(* CODESYS project OC_Profinet.library
   DefaultNamespace: OC_Profinet
   Description: Open Commissioning Library for Profinet devices
   Author: SpiraTec AG
   Title: OC_Profinet
   Version: 1.0.1
   Company: Open Commissioning
   Placeholder: OC_Profinet

Project tree, tasks and I/O mapping:
  libraries: OC_Core, * (Open Commissioning); OC_Profisafe, * (Open Commissioning); Tc2_Math, * (Beckhoff Automation GmbH); Tc2_Standard, * (Beckhoff Automation GmbH); Tc2_System, * (Beckhoff Automation GmbH); Tc2_Utilities, * (Beckhoff Automation GmbH); Tc3_Module, * (Beckhoff Automation GmbH); TcUnit, * (www.tcunit.org)
  Common/
    ProfidriveGSM/
      data type E_ProfidriveGSM_State
      function block FB_ProfidriveGSM [ST]: eState, S0_Disabled, S1_SwitchingOnInhibited, S2_ReadyForSwitchingOn, S3_SwitchedOn, S4_Operation, S51_RampStop, S52_QuickStop
      data type ST_ProfidriveGSM_Control
      data type ST_ProfidriveGSM_Status
    ProfidriveParamInterpreter/
      data type E_ProfidriveParam_Format
      function block FB_ProfidriveParamInterpreter [ST]: FormatSize, FormatType, MakeResponse, Reset
      data type ST_ProfidriveParam
      data type ST_ProfidriveParam_Set
    Utils/
      function F_CalcCrc16 [ST]
  Devices/
    Profidrive_Telegram1/
      function block FB_Profidrive_Telegram1 [ST]: Cycle, GetControlData, InitRun, Operation, SetStatusData
      data type ST_Profidrive_Telegram1_Config
      data type ST_Profidrive_Telegram1_Control
      data type ST_Profidrive_Telegram1_Status
    SEW_MoviC_Position/
      data type E_SEW_MoviC_Position_OperationMode
      function block FB_SEW_MoviC_Position [ST]: Cycle, GetControlData, InitRun, Operation, Safety, SetStatusData
      data type ST_SEW_MoviC_Position_Config
      data type ST_SEW_MoviC_Position_Control
      data type ST_SEW_MoviC_Position_Status
    SEW_MoviC_Velocity/
      function block FB_SEW_MoviC_Velocity [ST]: Cycle, GetControlData, InitRun, Operation, Safety, SetStatusData
      data type ST_SEW_MoviC_Velocity_Config
      data type ST_SEW_MoviC_Velocity_Control
      data type ST_SEW_MoviC_Velocity_Status
    SEW_Movisafe_CSSx1a/
      function block FB_SEW_Movisafe_CSSx1a [ST]: bSTO, Cycle, GetControlData, InitRun, SetStatusData
      data type ST_SEW_Movisafe_CSSx1a_Config
      data type ST_SEW_Movisafe_CSSx1a_Control
      data type ST_SEW_Movisafe_CSSx1a_Status
    Siemens_RcvDp/
      function block FB_Siemens_RcvDp [ST]: Cycle, GetControlData, InitRun, SetStatusData, SimLogic
      data type ST_Siemens_RcvDp_Config
      data type ST_Siemens_RcvDp_Control
      data type ST_Siemens_RcvDp_DevData
      data type ST_Siemens_RcvDp_HstData
      data type ST_Siemens_RcvDp_Status
    Siemens_SendDp/
      function block FB_Siemens_SendDp [ST]: Cycle, GetControlData, InitRun, SetStatusData, SimLogic
      data type ST_Siemens_SendDp_Config
      data type ST_Siemens_SendDp_Control
      data type ST_Siemens_SendDp_DevData
      data type ST_Siemens_SendDp_HstData
      data type ST_Siemens_SendDp_Status
    interface I_SEW_Movisafe: bSTO
*)

// Common/ProfidriveGSM/E_ProfidriveGSM_State
{attribute 'qualified_only'}
{attribute 'strict'}
{attribute 'conditionalshow'}
TYPE E_ProfidriveGSM_State :
(
	S0_Disabled := 0,
	S1_SwitchingOnInhibited := 1,
	S2_ReadyForSwitchingOn := 2,
	S3_SwitchedOn := 3,
	S4_Operation := 4,
	S51_RampStop := 51,
	S52_QuickStop := 52
);
END_TYPE

// Common/ProfidriveGSM/ST_ProfidriveGSM_Control
(*
	Steuerwort 1 (STW1)
	Steuerwort 1 SIEMENS Telegramm 10x
	https://cache.industry.siemens.com/dl/files/665/109770665/att_1023132/v2/109770665_PROFIdrive_Statemachine_DOC_V10_de.pdf
*)
{attribute 'pack_mode' := '1'}
TYPE ST_ProfidriveGSM_Control :
STRUCT
	b0_On 							: BIT; 	//ON/OFF (OFF1)
	b1_CoastStop					: BIT; 	//The axis will not coast stop if this bit is set (OFF2)
	b2_QuickStop					: BIT; 	//The axis will not execute quick stop if this bit is set. Quick stop executes a controlled stop on the axis. (OFF3)
	b3_EnableOperation				: BIT; 	//The axis will enable and execute command if all preconditions are set. If a Wake and Shake procedure has to be executed as part of enabling, the transition to state "S4: Operation Enabled" is delayed until the procedure is finished.
	b4_Reserve						: BIT;	//Reserve
	b5_Reserve						: BIT;	//Reserve
	b6_Reserve						: BIT;	//Reserve
	b7_FaultAcknowledge				: BIT;	//Set this bit to reset faults on the drive.
	b8_Reserve						: BIT;	//Reserve
	b9_Reserve						: BIT;	//Reserve	
	b10_ControlPlc					: BIT;	//When not set, no command is accepted from the PLC.	
	b11_Reserved					: BIT;	//Reserve
	b12_Reserved					: BIT;	//Reserve
	b13_Reserved					: BIT;	//Reserve
	b14_Reserved					: BIT;	//Reserve
	b15_Reserved					: BIT;	//Reserve
END_STRUCT
END_TYPE

// Common/ProfidriveGSM/ST_ProfidriveGSM_Status
(*
	Zustandswort 1 (ZSW1)
	Zustandswort 1 SIEMENS Telegramm 10x
	https://cache.industry.siemens.com/dl/files/665/109770665/att_1023132/v2/109770665_PROFIdrive_Statemachine_DOC_V10_de.pdf
*)

{attribute 'pack_mode' := '1'}
TYPE ST_ProfidriveGSM_Status :
STRUCT
	b0_ReadyToSwitchOn 				: BIT; 	//Ready to switch on
	b1_ReadyForOperation			: BIT; 	//Ready for operation
	b2_OperationEnabled				: BIT; 	//Operation enabled
	b3_FaultPresent					: BIT; 	//A fault is present on the axis
	b4_CoastStop 					: BIT;	//No coast stop is executed (No OFF2 is active)
	b5_QuickStop					: BIT;	//No quick stop is executed (No OFF3 is active)
	b6_SwitchingOnInhibited			: BIT;	//Switch-on inhibit Switching on again is only possible through OFF1 and subsequent ON.
	b7_WarningPresent				: BIT;	//Warning present. The drive is operating. No acknowledgment required
	b8_Reserve						: BIT;	//Reserve
	b9_ControlRequested				: BIT;	//Control requested by the master
	b10_Reserved					: BIT;	//Reserve
	b11_Reserved					: BIT;	//Reserve
	b12_Reserved					: BIT;	//Reserve
	b13_Reserved					: BIT;	//Reserve
	b14_Reserved					: BIT;	//Reserve
	b15_Reserved					: BIT;	//Reserve
END_STRUCT
END_TYPE

// Common/ProfidriveParamInterpreter/E_ProfidriveParam_Format
{attribute 'qualified_only'}
{attribute 'strict'}
{attribute 'conditionalshow'}
TYPE E_ProfidriveParam_Format :
(
	UNKNOWN := 0,
	INT8	:= 2,
	INT16	:= 3,
	INT32	:= 4,
	UINT8	:= 5,
	UINT16	:= 6,
	UINT32	:= 7,
	FLOAT	:= 8,
	ZERO	:= 64,
	BYTE_	:= 65,
	WORD_	:= 66,
	DWORD_	:= 67,
	ERROR	:= 68
) BYTE;
END_TYPE

// Common/ProfidriveParamInterpreter/ST_ProfidriveParam
{attribute 'conditionalshow'}
TYPE ST_ProfidriveParam :
STRUCT
	nAttribute	: BYTE;
	nNumber		: UINT;
	nSubIndex	: UINT;
	nElements	: BYTE;
	nFormat		: E_ProfidriveParam_Format;
	aValue		: ARRAY[0..234] OF BYTE;
END_STRUCT
END_TYPE

// Common/ProfidriveParamInterpreter/ST_ProfidriveParam_Set
{attribute 'conditionalshow'}
TYPE ST_ProfidriveParam_Set :
	ARRAY[0..22] OF ST_ProfidriveParam; 
END_TYPE

// Devices/Profidrive_Telegram1/ST_Profidrive_Telegram1_Config
TYPE ST_Profidrive_Telegram1_Config :
STRUCT
	bForceMode					: BOOL; //Ignore process data from fieldbus.
	bSwapProcessData			: BOOL; //Reverse process data byte order from/to fieldbus.
	fRampDownTimeCoastStop 		: REAL := 1.0;		//Coast stop deceleration time in s
	bControlRequested			: BOOL := TRUE;
	bOutputVelocity				: BOOL := TRUE;		//TRUE: TargetValue = Velocity, FALSE: TargetValue = Position
	fP1058						: REAL := 150.0;	//JOG 1 velocity in rotation/s
	fP1059						: REAL := -150.0;	//JOG 1 velocity in rotation/s
	fP1120						: REAL := 2.0;		//Default acceleration time in s
	fP1121						: REAL := 2.0;		//Default deceleration time in s
	fP1135						: REAL := 1.0;		//Ramp down time quick stop in s
	fP2000						: REAL := 3000;		//Velocity in rotation/s when targeting 16#4000
	nR0035						: REAL := 60.0; 	//Temperature in degree celcius	
END_STRUCT
END_TYPE

// Devices/Profidrive_Telegram1/ST_Profidrive_Telegram1_Control
TYPE ST_Profidrive_Telegram1_Control :
STRUCT
	b0_Off1								: BOOL;	//STW1_0	0 = OFF1 (braking with ramp-function generator, then pulse suppression & ready for switching on) | 0 → 1 = ON (pulses can be enabled)
	b1_Off2								: BOOL;	//STW1_1	0 = OFF2 (immediate pulse suppression and switching on inhibited) | 1 = No OFF2 (enable is possible)
	b2_Off3								: BOOL;	//STW1_2	0 = OFF3 (braking with the OFF3 ramp p1135, then pulse suppression and switching on inhibited) | 1 = No OFF3 (enable possible) 
	b3_EnableOperation					: BOOL;	//STW1_3	0 = Inhibit operation (suppress pulses) | 1 = Enable operation (pulses can be enabled) 
	b4_OperatingCondition				: BOOL;	//STW1_4	0 = Inhibit ramp-function generator (set the ramp-function generator output to zero) | 1 = Operating condition (the ramp-function generator can be enabled)
	b5_ContinueRampFunctionGenerator	: BOOL;	//STW1_5	0 = Freeze ramp-function generator (freeze the ramp-function generator output) | 1 = Continue ramp-function generator 
	b6_EnableSetpoint  					: BOOL;	//STW1_6	0 = Inhibit setpoint (set the ramp-function generator input to zero) | 1 = Enable setpoint 
	b7_AcknowledgeFaults				: BOOL;	//STW1_7	0 → 1: = Acknowledge faults	                            
	b8_Jog1								: BOOL;	//STW1_8	1 = Jog 1 signal source
	b9_Jog2								: BOOL;	//STW1_9	1 = Jog 2 signal source
	b10_ControlByPlc					: BOOL;	//STW1_10	1 = Control by PLC
	b11_SetpointInversion				: BOOL;	//STW1_11	1 = Setpoint inversion
	b12_Reserved						: BOOL;	//STW1_12	Reserved
	b13_PotentiometerSetpointRaise		: BOOL;	//STW1_13	1 = Motorized potentiometer setpoint raise
	b14_PotentiometerSetpointLower		: BOOL;	//STW1_14	1 = Motorized potentiometer setpoint lower
	b15_Reserved						: BOOL;	//STW1_15	Reserved	
	nTargetVelocity						: INT;
END_STRUCT
END_TYPE

// Devices/Profidrive_Telegram1/ST_Profidrive_Telegram1_Status
TYPE ST_Profidrive_Telegram1_Status :
STRUCT
	b0_ReadyForSwitchingOn				: BOOL; // ZSW1_0	1 = Ready for switching on
	b1_ReadyForOperation				: BOOL; // ZSW1_1	1 = Ready for operation
	b2_OperationEnabled					: BOOL; // ZSW1_2	1 = Operation enabled
	b3_FaultPresent						: BOOL; // ZSW1_3	1 = Fault present
	b4_NoCoastDownActive				: BOOL; // ZSW1_4	1 = No coast down active (OFF2 inactive)
	b5_NoQuickStopActive				: BOOL; // ZSW1_5	1 = No quick stop active (OFF3 inactive)
	b6_SwitchingOnInhibited				: BOOL; // ZSW1_6	1 = Switching on inhibited active
	b7_AlarmPresent						: BOOL; // ZSW1_7	1 = Alarm present                        	
	b8_DeviationWithinTolerance			: BOOL; // ZSW1_8	1 = Speed setpoint - actual value deviation within tolerance t_off
	b9_ControlRequested					: BOOL; // ZSW1_9	1 = Control requested        
	b10_RpmCompValueReachedOrExceeded	: BOOL; // ZSW1_10	1 = f or n comparison value reached/exceeded  
	b11_TorqueOrPowerLimitNotReached	: BOOL; // ZSW1_11	1 = I, M, or P limit not reached     
	b12_OpenHoldingBrake 				: BOOL; // ZSW1_12	1 = Open the holding brake      
	b13_NoOvertempAlarm					: BOOL; // ZSW1_13	1 = No motor overtemperature alarm      
	b14_MotorRotatesForwards			: BOOL; // ZSW1_14	1 = Motor rotates forwards (n_act >= 0) | 0 = Motor rotates backwards (n_act < 0)   
	b15_NoAlarmNoOvertempPowerUnit		: BOOL; // ZSW1_15	1 = No alarm, thermal overload, power unit  
	nVelocity							: INT;
END_STRUCT
END_TYPE

// Devices/SEW_MoviC_Position/E_SEW_MoviC_Position_OperationMode
{attribute 'qualified_only'}
TYPE E_SEW_MoviC_Position_OperationMode :
(
	Jog					:= 100, //Position controlled jogging
	JogNoEnc			:= 101, //Speed controlled jogging
	SpeedControl		:= 200, //Speed control
	ReferenceParam		:= 300, //Reference travel, offset via parameter
	ReferenceBus		:= 301, //Reference travel, offset via fieldbus
	PositionAbs			:= 400, //Absolute position control
	PositionRel			:= 401, //Relative position control
	PositionModPos		:= 402, //Modulo position control, positive
	PositionModNeg		:= 403, //Modulo position control, negative
	PositionModShort	:= 404, //Modulo position control, shortest distance
	EnergyOptimized		:= 1200, //Energieoptimiertes Positionieren
	MechanicsOptimized	:= 1210	 //Mechanikoptimiertes Positionieren
)INT;
END_TYPE

// Devices/SEW_MoviC_Position/ST_SEW_MoviC_Position_Config
TYPE ST_SEW_MoviC_Position_Config :
STRUCT
	bForceMode				: BOOL; //Ignore process data from fieldbus.
	bSwapProcessData		: BOOL; //Reverse process data byte order from/to fieldbus.
	nSoftwareLimitMin		: DINT := -2147483648;	//Position limit minimum in LU
	nSoftwareLimitMax		: DINT := 2147483647;	//Position limit maximum in LU
	nReferencePos			: DINT := 0;			//Reference position in LU when using mode 300
	fDecCoastStop			: REAL := 1000.0;		//Deceleration for coast/brake stop in LU/s^2
	fDecEstop				: REAL := 100.0;		//Deceleration for emergency stop in LU/s^2
	fDecelerationLimit		: REAL := 100.0;		//Decceleration limit (bus stop) in LU/s^2
	fRatioVelocity			: REAL := 1.0;			//Ratio for setpoint velocity
	fRatioAccDec			: REAL := 1.0;			//Ratio for setpoint acceleration/deceleration
	fRatioPosition			: REAL := 1.0;			//Ratio for position output
	nJerk					: INT  := 0;			//Jerk from 0 to 100%
	fPositionOffset			: REAL := 0;
	fInitPosition			: REAL := 0;
	fResolution				: REAL := 0.1;
END_STRUCT
END_TYPE

// Devices/SEW_MoviC_Position/ST_SEW_MoviC_Position_Control
{attribute 'pack_mode' := '1'}
TYPE ST_SEW_MoviC_Position_Control :
STRUCT
    b0_EnableEStop 					: BIT;	//0  1 = enable, 0 = emergency stop
    b1_EnableBusStop 				: BIT;	//1  1 = enable, 0 = stop at application limits
    b2_Reserved2 					: BIT;	//2
    b3_ReleaseBrake 				: BIT;	//3  only needed if function is activated
    b4_JoggingCW 					: BIT;	//4  jog positive
    b5_JoggingCCW 					: BIT;	//5  jog negative
    b6_AcceptRelativePosition 		: BIT;	//6  apply relative target pos only in relative pos mode
    b7_StartStop 					: BIT;	//7  1 = start movement in all modes except jog, 0 = deceleration to speed 0
    b8_ErrorReset 					: BIT;	//8  reset fault messages
    b9_Reserved9 					: BIT;	//9
    b10_ActivateDriveTrain2 		: BIT;	//10  0 = drive train 1 selected, 1 = drive train 2 selected
    b11_Reserved11 					: BIT;	//11
    b12_DisableSoftwareLimits 		: BIT;	//12  0 = software limit activated, 1 = software limit deactivated
    b13_ActivateInhibit 			: BIT;	//13  1 = output stage inhibit activated -> motor coasts to halt or brake is applied, 0 = output stage can be enabled
    b14_ActivateStandByMode 		: BIT;	//14  1 = activated, can only be activated when output stage is inhibited (bActivateInhibit = 1)
    b15_MovikitHeartbeat 			: BIT;	//15  Heartbeat trigger
	nSetpointSpeed					: INT;	//16..31 
	nSetpointAcceleration			: INT;	//32..47
	nSetpointDeceleration			: INT;	//48..63
	nDigitalOutputs					: WORD;	//64..79
	nTargetApplicationMode			: E_SEW_MoviC_Position_OperationMode; //80..95
	nTargetPosition					: DINT;	//96..127
END_STRUCT
END_TYPE

// Devices/SEW_MoviC_Position/ST_SEW_MoviC_Position_Status
{attribute 'pack_mode' := '1'}
TYPE ST_SEW_MoviC_Position_Status :
STRUCT
	b0_InverterReady					: BIT;	//0  1 = Ready
	b1_STOInactive						: BIT;	//1  1 = STO inactive
	b2_PowerStageOn						: BIT;	//2  1 = Output stage enable
	b3_BrakeReleased					: BIT;	//3  1 = Brake released
	b4_MotorTurning						: BIT;	//4  1 = Motor running
	b5_DriveReferenced					: BIT;	//5  1 = Active drive referenced
	b6_SetpointsActive					: BIT;	//6  1 = New relative position applied
	b7_TargetpositionReached			: BIT;	//7  1 = In position
	b8_ErrorActive						: BIT;	//8  1 = Fault
	b9_WarningActive					: BIT;	//9  1 = Warning
	b10_DriveTrain2Active				: BIT;	//10  1 = Drive train 2 active
	b11_SpeedSetpointReached			: BIT;	//11  1 = "Setpoint/actual speed comparison active" signal
	b12_SoftwareLimitsDisabled			: BIT;	//12  1 = Software limit switches inactive
	b13_OutputStageInhibit 				: BIT;	//13  1 = Output stage inhibit 
	b14_StandByModeActive				: BIT;	//14  1 = Standby mode active
	b15_MovikitHeartbeat				: BIT;	//15  Heartbeat trigger mirror
	nActualSpeed						: INT;	//16..31
	nActualStatus						: WORD;	//32..47
	nActualTorque						: INT;	//48..63
	nDigitalInputs						: WORD;	//64..79
	nActualApplicationMode				: E_SEW_MoviC_Position_OperationMode; //80..95
	nActualPosition						: DINT;	//96..127 
END_STRUCT
END_TYPE

// Devices/SEW_MoviC_Velocity/ST_SEW_MoviC_Velocity_Config
TYPE ST_SEW_MoviC_Velocity_Config :
STRUCT
	bForceMode				: BOOL; //Ignore process data from fieldbus.
	bSwapProcessData		: BOOL; //Reverse process data byte order from/to fieldbus.
	nSoftwareLimitMin		: DINT := -2147483648;	//Position limit minimum in LU
	nSoftwareLimitMax		: DINT := 2147483647;	//Position limit maximum in LU
	nReferencePos			: DINT := 0;			//Reference position in LU when using mode 300
	fDecCoastStop			: REAL := 1000.0;		//Deceleration for coast/brake stop in LU/s^2
	fDecEstop				: REAL := 100.0;		//Deceleration for emergency stop in LU/s^2
	fDecelerationLimit		: REAL := 100.0;		//Decceleration limit (bus stop) in LU/s^2
	fRatioVelocity			: REAL := 1.0;			//Ratio for setpoint velocity
	fRatioAccDec			: REAL := 1.0;			//Ratio for setpoint acceleration/deceleration
	fRatioPosition			: REAL := 1.0;			//Ratio for position output
	nJerk					: INT  := 0;			//Jerk from 0 to 100%
	fPositionOffset			: REAL := 0;
	fInitPosition			: REAL := 0;
	fResolution				: REAL := 0.1;
	bOutputVelocity			: BOOL := TRUE;			//TRUE: TargetValue = Velocity, FALSE: TargetValue = Position
END_STRUCT
END_TYPE

// Devices/SEW_MoviC_Velocity/ST_SEW_MoviC_Velocity_Control
TYPE ST_SEW_MoviC_Velocity_Control :
STRUCT
    b0_EnableEStop 					: BIT;	//0  1 = enable, 0 = emergency stop
    b1_EnableBusStop 				: BIT;	//1  1 = enable, 0 = stop at application limits
    b2_Reserved2 					: BIT;	//2
    b3_ReleaseBrake 				: BIT;	//3  only needed if function is activated
    b4_JoggingCW 					: BIT;	//4  jog positive
    b5_JoggingCCW 					: BIT;	//5  jog negative
    b6_AcceptRelativePosition 		: BIT;	//6  apply relative target pos only in relative pos mode
    b7_StartStop 					: BIT;	//7  1 = start movement in all modes except jog, 0 = deceleration to speed 0
    b8_ErrorReset 					: BIT;	//8  reset fault messages
    b9_Reserved9 					: BIT;	//9
    b10_ActivateDriveTrain2 		: BIT;	//10  0 = drive train 1 selected, 1 = drive train 2 selected
    b11_Reserved11 					: BIT;	//11
    b12_DisableSoftwareLimits 		: BIT;	//12  0 = software limit activated, 1 = software limit deactivated
    b13_ActivateInhibit 			: BIT;	//13  1 = output stage inhibit activated -> motor coasts to halt or brake is applied, 0 = output stage can be enabled
    b14_ActivateStandByMode 		: BIT;	//14  1 = activated, can only be activated when output stage is inhibited (bActivateInhibit = 1)
    b15_MovikitHeartbeat 			: BIT;	//15  Heartbeat trigger
	nSetpointSpeed					: INT;	//16..31 
	nSetpointAcceleration			: INT;	//32..47
	nSetpointDeceleration			: INT;	//48..63
	nDigitalOutputs					: WORD;	//64..79	
END_STRUCT
END_TYPE

// Devices/SEW_MoviC_Velocity/ST_SEW_MoviC_Velocity_Status
{attribute 'pack_mode' := '1'}
TYPE ST_SEW_MoviC_Velocity_Status :
STRUCT
	b0_InverterReady					: BIT;	//0  1 = Ready
	b1_STOInactive						: BIT;	//1  1 = STO inactive
	b2_PowerStageOn						: BIT;	//2  1 = Output stage enable
	b3_BrakeReleased					: BIT;	//3  1 = Brake released
	b4_MotorTurning						: BIT;	//4  1 = Motor running
	b5_DriveReferenced					: BIT;	//5  1 = Active drive referenced
	b6_SetpointsActive					: BIT;	//6  1 = New relative position applied
	b7_TargetpositionReached			: BIT;	//7  1 = In position
	b8_ErrorActive						: BIT;	//8  1 = Fault
	b9_WarningActive					: BIT;	//9  1 = Warning
	b10_DriveTrain2Active				: BIT;	//10  1 = Drive train 2 active
	b11_SpeedSetpointReached			: BIT;	//11  1 = "Setpoint/actual speed comparison active" signal
	b12_SoftwareLimitsDisabled			: BIT;	//12  1 = Software limit switches inactive
	b13_OutputStageInhibit 				: BIT;	//13  1 = Output stage inhibit 
	b14_StandByModeActive				: BIT;	//14  1 = Standby mode active
	b15_MovikitHeartbeat				: BIT;	//15  Heartbeat trigger mirror
	nActualSpeed						: INT;	//16..31
	nActualStatus						: WORD;	//32..47
	nActualTorque						: INT;	//48..63
	nDigitalInputs						: WORD;	//64..79	
END_STRUCT
END_TYPE

// Devices/SEW_Movisafe_CSSx1a/ST_SEW_Movisafe_CSSx1a_Config
TYPE ST_SEW_Movisafe_CSSx1a_Config :
STRUCT	
	bForceMode			: BOOL; //Ignore process data from fieldbus.
	bSwapProcessData	: BOOL; //Reverse process data byte order from/to fieldbus.
END_STRUCT
END_TYPE

// Devices/SEW_Movisafe_CSSx1a/ST_SEW_Movisafe_CSSx1a_Control
{attribute 'pack_mode' := '1'}
TYPE ST_SEW_Movisafe_CSSx1a_Control :
STRUCT
	b0_0_STO			: BIT; //0.0  Sicher abgeschaltetes Drehmoment
	b0_1_SLI			: BIT; //0.1  Freigabe SLI (Sicher begrenztes Schrittmaß)
	b0_2_SBT			: BIT; //0.2  Freigabe SBT (Sicherer Bremsentest)
	b0_3_Reserved		: BIT; //0.3  Reserve
	b0_4_MutingEncErr	: BIT; //0.4  Muting Geber anwählen
	b0_5_TestModeActice	: BIT; //0.5  Test Modus der Antriebssicherheitsfunktion anwählen
	b0_6_AckFDI			: BIT; //0.6  Quittierung der verriegelten Digitaleingänge
	b0_7_AckError		: BIT; //0.7  Quittierung der Fehler Sicherheitskarte
	b1_0_F_DO0			: BIT; //1.0  F-DO 00 Digitaler Ausgang 0
	b1_1_F_DO1			: BIT; //1.1  F-DO 01 Digitaler Ausgang 1
	b1_2_Reserved		: BIT; //1.2  Reserve
	b1_3_Reserved		: BIT; //1.3  Reserve
	b1_4_Reserved		: BIT; //1.4  Reserve
	b1_5_Reserved		: BIT; //1.5  Reserve
	b1_6_Reserved		: BIT; //1.6  Reserve
	b1_7_Reserved		: BIT; //1.7  Reserve
	b2_0_SOS1			: BIT; //2.0  SOS1 deaktivieren (Sicherer Betriebshalt)
	b2_1_Reserved		: BIT; //2.1  Reserve
	b2_2_SSx1			: BIT; //2.2  Antriebssicherheitsfunktion SSx1 deaktivieren
	b2_3_SSx2			: BIT; //2.3  Antriebssicherheitsfunktion SSx2 deaktivieren
	b2_4_SDI1			: BIT; //2.4  SDI 1 deaktivieren (Sichere Bewegungsrichtung)
	b2_5_SDI2			: BIT; //2.5  SDI 2 deaktivieren (Sichere Bewegungsrichtung)
	b2_6_SLI1			: BIT; //2.6  SLI 1 deaktivieren (Sicher begrenztes Schrittmaß)
	b2_7_SLI2			: BIT; //2.7  SLI 2 deaktivieren (Sicher begrenztes Schrittmaß)
	b3_0_SLS1			: BIT; //3.0  SLS 1 deaktivieren (Sicher begrenzte Geschwindigkeit)
	b3_1_SLS2			: BIT; //3.1  SLS 2 deaktivieren (Sicher begrenzte Geschwindigkeit)
	b3_2_SLS3			: BIT; //3.2  SLS 3 deaktivieren (Sicher begrenzte Geschwindigkeit)
	b3_3_SLS4			: BIT; //3.3  SLS 4 deaktivieren (Sicher begrenzte Geschwindigkeit)
	b3_4_SSR1			: BIT; //3.4  SSR 1 deaktivieren (Sicherer Geschwindigkeitsbereich)
	b3_5_SSR2			: BIT; //3.5  SSR 2 deaktivieren (Sicherer Geschwindigkeitsbereich)
	b3_6_Reserved		: BIT; //3.6  Reserve
	b3_7_Reserved		: BIT; //3.7  Reserve
	b4_0_SLA1			: BIT; //4.0  SLA 1 deaktivieren (Sicher begrenzte Beschleunigung)
	b4_1_SLA2			: BIT; //4.1  SLA 2 deaktivieren (Sicher begrenzte Beschleunigung)
	b4_2_Reserved		: BIT; //4.2  Reserve
	b4_3_Reserved		: BIT; //4.3  Reserve
	b4_4_Reserved		: BIT; //4.4  Reserve
	b4_5_Reserved		: BIT; //4.5  Reserve
	b4_6_Reserved		: BIT; //4.6  Reserve
	b4_7_Reserved		: BIT; //4.7  Reserve
END_STRUCT
END_TYPE

// Devices/SEW_Movisafe_CSSx1a/ST_SEW_Movisafe_CSSx1a_Status
{attribute 'pack_mode' := '1'}
TYPE ST_SEW_Movisafe_CSSx1a_Status :
STRUCT
	b0_0_STOActive		: BIT; //0.0  Sicher abgeschaltetes Drehmoment
	b0_1_ASFDiag		: BIT; //0.1  Mindestens eine Antriebssicherheitsfunktion hat eine Grenze überschritten
	b0_2_SBTActive		: BIT; //0.2  Bremsentest ist aktiv
	b0_3_InputDataValid	: BIT; //0.3  Alle Prozesswerte der F-DI enthalten aktuelle Werte
	b0_4_MutingEncErr	: BIT; //0.4  Geber Muting Funktion ist aktive
	b0_5_TestModeActive	: BIT; //0.5  Test Modus der Antriebssicherheitsfunktion ist aktive
	b0_6_Warning		: BIT; //0.6  Warnung in der Safety-option
	b0_7_ErrorState		: BIT; //0.7  Fehler in der Safety-option
	b1_0_F_DI0			: BIT; //1.0  Zustand digitaler Eingang 1
	b1_1_F_DI1			: BIT; //1.1  Zustand digitaler Eingang 2
	b1_2_F_DI2			: BIT; //1.2  Zustand digitaler Eingang 3
	b1_3_F_DI3			: BIT; //1.3  Zustand digitaler Eingang 4
	b1_4_Reserved		: BIT; //1.4  Reserve
	b1_5_Reserved		: BIT; //1.5  Reserve
	b1_6_Reserved		: BIT; //1.6  Reserve
	b1_7_Reserved		: BIT; //1.7  Reserve
	b2_0_SOS1			: BIT; //2.0  SOS1 ist aktiviert (Sicherer Betriebshalt)
	b2_1_Reserved		: BIT; //2.1  Reserve
	b2_2_SSx1			: BIT; //2.2  SSx1  ist aktiviert
	b2_3_SSx2			: BIT; //2.3  SSx2 ist aktiviert
	b2_4_SDI1			: BIT; //2.4  SDI 1  ist aktiviert (Sichere Bewegungsrichtung)
	b2_5_SDI2			: BIT; //2.5  SDI 2  ist aktiviert (Sichere Bewegungsrichtung)
	b2_6_SLI1			: BIT; //2.6  SLI 1  ist aktiviert (Sicher begrenztes Schrittmaß)
	b2_7_SLI2			: BIT; //2.7  SLI 2  ist aktiviert (Sicher begrenztes Schrittmaß)
	b3_0_SLS1			: BIT; //3.0  SLS 1  ist aktiviert (Sicher begrenzte Geschwindigkeit)
	b3_1_SLS2			: BIT; //3.1  SLS 2  ist aktiviert (Sicher begrenzte Geschwindigkeit)
	b3_2_SLS3			: BIT; //3.2  SLS 3  ist aktiviert (Sicher begrenzte Geschwindigkeit)
	b3_3_SLS4			: BIT; //3.3  SLS 4  ist aktiviert (Sicher begrenzte Geschwindigkeit)
	b3_4_SSR1			: BIT; //3.4  SSR 1  ist aktiviert (Sicherer Geschwindigkeitsbereich)
	b3_5_SSR2			: BIT; //3.5  SSR 2  ist aktiviert (Sicherer Geschwindigkeitsbereich)
	b3_6_Reserved		: BIT; //3.6  Reserve
	b3_7_Reserved		: BIT; //3.7  Reserve
	b4_0_SLA1			: BIT; //4.0  SLA 1  ist aktiviert (Sicher begrenzte Beschleunigung)
	b4_1_SLA2			: BIT; //4.1  SLA 2  ist aktiviert (Sicher begrenzte Beschleunigung)
	b4_2_SSM1			: BIT; //4.2  SSM 1  ist aktiviert (Sichere Geschwindigkeitsüberwachung)
	b4_3_SSM2			: BIT; //4.3  SSM 2  ist aktiviert (Sichere Geschwindigkeitsüberwachung)
	b4_4_SSM3			: BIT; //4.4  SSM 3  ist aktiviert (Sichere Geschwindigkeitsüberwachung)
	b4_5_SSM4			: BIT; //4.5  SSM 4  ist aktiviert (Sichere Geschwindigkeitsüberwachung)
	b4_6_Reserved		: BIT; //4.6  Reserve
	b4_7_Reserved		: BIT; //4.7  Reserve
	b5_0_Reserved		: BIT; //5.0  Reserve
	b5_1_Reserved		: BIT; //5.1  Reserve
	b5_2_Reserved		: BIT; //5.2  Reserve
	b5_3_Reserved		: BIT; //5.3  Reserve
	b5_4_Reserved		: BIT; //5.4  Reserve
	b5_5_Reserved		: BIT; //5.5  Reserve
	b5_6_Reserved		: BIT; //5.6  Reserve
	b5_7_Reserved		: BIT; //5.7  Reserve
END_STRUCT
END_TYPE

// Devices/Siemens_RcvDp/ST_Siemens_RcvDp_Config
TYPE ST_Siemens_RcvDp_Config :
STRUCT
	bForceMode			: BOOL; //Ignore process data from fieldbus.
	bSwapProcessData	: BOOL; //Reverse process data byte order from/to fieldbus.
	nDpDpId			 	: UINT := 0;
	fTimeout		 	: REAL := 0.5;
	bAutoAckRei			: BOOL := TRUE;
END_STRUCT
END_TYPE

// Devices/Siemens_RcvDp/ST_Siemens_RcvDp_Control
{attribute 'pack_mode' := '1'}
TYPE ST_Siemens_RcvDp_Control :
STRUCT
	nRcvBoolData			: WORD;
	nRcvInt00				: INT;
	nRcvInt01				: INT;
	nRcvData				: WORD;
	nRcvSequenceNumber		: WORD;
	nRcvCrc					: WORD;
END_STRUCT
END_TYPE

// Devices/Siemens_RcvDp/ST_Siemens_RcvDp_DevData
TYPE ST_Siemens_RcvDp_DevData :
STRUCT
	bAckRei		: BOOL;
	bSub00		: BOOL;
	bSub01		: BOOL;
	bSub02		: BOOL;
	bSub03		: BOOL;
	bSub04		: BOOL;
	bSub05		: BOOL;
	bSub06		: BOOL;
	bSub07		: BOOL;
	bSub08		: BOOL;
	bSub09		: BOOL;
	bSub10		: BOOL;
	bSub11		: BOOL;
	bSub12		: BOOL;
	bSub13		: BOOL;
	bSub14		: BOOL;
	bSub15		: BOOL;
	nSub00		: INT;
	nSub01		: INT;
END_STRUCT
END_TYPE

// Devices/Siemens_RcvDp/ST_Siemens_RcvDp_HstData
TYPE ST_Siemens_RcvDp_HstData :
STRUCT
	bError		: BOOL;
	bSubsOn		: BOOL;
	bRcv00		: BOOL;
	bRcv01		: BOOL;
	bRcv02		: BOOL;
	bRcv03		: BOOL;
	bRcv04		: BOOL;
	bRcv05		: BOOL;
	bRcv06		: BOOL;
	bRcv07		: BOOL;
	bRcv08		: BOOL;
	bRcv09		: BOOL;
	bRcv10		: BOOL;
	bRcv11		: BOOL;
	bRcv12		: BOOL;
	bRcv13		: BOOL;
	bRcv14		: BOOL;
	bRcv15		: BOOL;
	nRcv00		: INT;
	nRcv01		: INT;
END_STRUCT
END_TYPE

// Devices/Siemens_RcvDp/ST_Siemens_RcvDp_Status
{attribute 'pack_mode' := '1'}
TYPE ST_Siemens_RcvDp_Status :
STRUCT
	nSendData				: WORD;
	nSendSequenceNumber		: WORD;	
	nSendCrc				: WORD;
END_STRUCT
END_TYPE

// Devices/Siemens_SendDp/ST_Siemens_SendDp_Config
TYPE ST_Siemens_SendDp_Config :
STRUCT
	bForceMode			: BOOL; //Ignore process data from fieldbus.
	bSwapProcessData	: BOOL; //Reverse process data byte order from/to fieldbus.
	nDpDpId			 	: UINT := 0;
	fTimeout		 	: REAL := 0.5;
END_STRUCT
END_TYPE

// Devices/Siemens_SendDp/ST_Siemens_SendDp_Control
TYPE ST_Siemens_SendDp_Control :
STRUCT
	nRcvData				: WORD;
	nRcvSequenceNumber		: WORD;	
	nRcvCrc					: WORD;
END_STRUCT
END_TYPE

// Devices/Siemens_SendDp/ST_Siemens_SendDp_DevData
TYPE ST_Siemens_SendDp_DevData :
STRUCT
	bSend00		: BOOL;
	bSend01		: BOOL;
	bSend02		: BOOL;
	bSend03		: BOOL;
	bSend04		: BOOL;
	bSend05		: BOOL;
	bSend06		: BOOL;
	bSend07		: BOOL;
	bSend08		: BOOL;
	bSend09		: BOOL;
	bSend10		: BOOL;
	bSend11		: BOOL;
	bSend12		: BOOL;
	bSend13		: BOOL;
	bSend14		: BOOL;
	bSend15		: BOOL;
	nSend00		: INT;
	nSend01		: INT;
END_STRUCT
END_TYPE

// Devices/Siemens_SendDp/ST_Siemens_SendDp_HstData
TYPE ST_Siemens_SendDp_HstData :
STRUCT
	bError		: BOOL;
	bSubsOn		: BOOL;
END_STRUCT
END_TYPE

// Devices/Siemens_SendDp/ST_Siemens_SendDp_Status
TYPE ST_Siemens_SendDp_Status :
STRUCT
	nSendBoolData			: WORD;
	nSendInt00				: INT;
	nSendInt01				: INT;
	nSendData				: WORD;
	nSendSequenceNumber		: WORD;
	nSendCrc				: WORD;
END_STRUCT
END_TYPE

// Common/ProfidriveGSM/FB_ProfidriveGSM
// Profidrive General State Machine
FUNCTION_BLOCK PUBLIC FB_ProfidriveGSM
VAR_INPUT
	bPowerOn					: BOOL := TRUE;
	bStandstill					: BOOL;
	nControl					: ST_ProfidriveGSM_Control;
END_VAR

VAR_OUTPUT
	nStatus						: ST_ProfidriveGSM_Status;
END_VAR

VAR	
	_eState 					: E_ProfidriveGSM_State := E_ProfidriveGSM_State.S1_SwitchingOnInhibited;
END_VAR

CASE _eState OF 
	E_ProfidriveGSM_State.S0_Disabled : S0_Disabled();
	E_ProfidriveGSM_State.S1_SwitchingOnInhibited : S1_SwitchingOnInhibited();
	E_ProfidriveGSM_State.S2_ReadyForSwitchingOn : S2_ReadyForSwitchingOn();
	E_ProfidriveGSM_State.S3_SwitchedOn : S3_SwitchedOn();
	E_ProfidriveGSM_State.S4_Operation : S4_Operation();
	E_ProfidriveGSM_State.S51_RampStop : S51_RampStop();
	E_ProfidriveGSM_State.S52_QuickStop : S52_QuickStop();
END_CASE

PROPERTY eState : E_ProfidriveGSM_State
GET
eState := _eState;
END_GET
SET
_eState := eState;
END_SET
END_PROPERTY

{ attribute 'hide' }
METHOD PROTECTED S0_Disabled
nStatus.b0_ReadyToSwitchOn 			:= FALSE;				
nStatus.b1_ReadyForOperation 		:= FALSE;				
nStatus.b2_OperationEnabled 		:= FALSE;					
nStatus.b3_FaultPresent 			:= FALSE;						
nStatus.b4_CoastStop 				:= FALSE;	 					
nStatus.b5_QuickStop 				:= FALSE;						
nStatus.b6_SwitchingOnInhibited 	:= FALSE;				
nStatus.b7_WarningPresent			:= FALSE;			
nStatus.b9_ControlRequested 		:= FALSE;	

(*to S1*)	
IF bPowerOn THEN
	_eState := E_ProfidriveGSM_State.S1_SwitchingOnInhibited;
END_IF
END_METHOD

{ attribute 'hide' }
METHOD INTERNAL S1_SwitchingOnInhibited
VAR_INPUT
END_VAR
nStatus.b0_ReadyToSwitchOn 		:= FALSE;				
nStatus.b1_ReadyForOperation 		:= FALSE;				
nStatus.b2_OperationEnabled 		:= FALSE;						
nStatus.b6_SwitchingOnInhibited 	:= TRUE;

(*to S2_ReadyForSwitchingOn*)	
IF NOT nControl.b0_On AND nControl.b1_CoastStop AND nControl.b2_QuickStop THEN
	_eState := E_ProfidriveGSM_State.S2_ReadyForSwitchingOn;
END_IF
END_METHOD

{ attribute 'hide' }
METHOD INTERNAL S2_ReadyForSwitchingOn
VAR_INPUT
END_VAR
nStatus.b0_ReadyToSwitchOn 		:= TRUE;				
nStatus.b1_ReadyForOperation 		:= FALSE;				
nStatus.b2_OperationEnabled 		:= FALSE;						
nStatus.b6_SwitchingOnInhibited 	:= FALSE;

(*to S1_SwitchingOnInhibited*)	
IF NOT nControl.b1_CoastStop OR NOT nControl.b2_QuickStop THEN
	_eState := E_ProfidriveGSM_State.S1_SwitchingOnInhibited;
	RETURN;
END_IF

(*to S3_SwitchedOn*)	
IF nControl.b0_On THEN
	_eState := E_ProfidriveGSM_State.S3_SwitchedOn;
END_IF
END_METHOD

{ attribute 'hide' }
METHOD INTERNAL S3_SwitchedOn
VAR_INPUT
END_VAR
nStatus.b0_ReadyToSwitchOn 		:= TRUE;				
nStatus.b1_ReadyForOperation 		:= TRUE;				
nStatus.b2_OperationEnabled 		:= FALSE;						
nStatus.b6_SwitchingOnInhibited 	:= FALSE;

(*to S1_SwitchingOnInhibited*)	
IF NOT nControl.b1_CoastStop OR NOT nControl.b2_QuickStop THEN
	_eState := E_ProfidriveGSM_State.S1_SwitchingOnInhibited;
	RETURN;
END_IF

(*to S2_ReadyForSwitchingOn*)	
IF NOT nControl.b0_On THEN
	_eState := E_ProfidriveGSM_State.S2_ReadyForSwitchingOn;
	RETURN;
END_IF

(*to S4_Operation*)	
IF nControl.b3_EnableOperation THEN
	_eState := E_ProfidriveGSM_State.S4_Operation;
END_IF
END_METHOD

{ attribute 'hide' }
METHOD INTERNAL S4_Operation
VAR_INPUT
END_VAR
nStatus.b0_ReadyToSwitchOn 		:= TRUE;				
nStatus.b1_ReadyForOperation 		:= TRUE;				
nStatus.b2_OperationEnabled 		:= TRUE;					
nStatus.b6_SwitchingOnInhibited 	:= FALSE;

(*to S1_SwitchingOnInhibited*)	
IF NOT nControl.b1_CoastStop THEN
	_eState := E_ProfidriveGSM_State.S1_SwitchingOnInhibited;
	RETURN;
END_IF

(*to S52_QuickStop*)	
IF NOT nControl.b2_QuickStop THEN
	_eState := E_ProfidriveGSM_State.S52_QuickStop;
	RETURN;
END_IF

(*to S51_RampStop*)	
IF NOT nControl.b0_On THEN
	_eState := E_ProfidriveGSM_State.S51_RampStop;
	RETURN;
END_IF

(*to S3_SwitchedOn*)	
IF NOT nControl.b3_EnableOperation THEN
	_eState := E_ProfidriveGSM_State.S3_SwitchedOn;
END_IF
END_METHOD

{ attribute 'hide' }
METHOD INTERNAL S51_RampStop
VAR_INPUT
END_VAR
nStatus.b0_ReadyToSwitchOn 		:= TRUE;				
nStatus.b1_ReadyForOperation 		:= TRUE;				
nStatus.b2_OperationEnabled 		:= FALSE;					
nStatus.b6_SwitchingOnInhibited 	:= FALSE;

(*to S1_SwitchingOnInhibited*)	
IF NOT nControl.b1_CoastStop THEN
	_eState := E_ProfidriveGSM_State.S1_SwitchingOnInhibited;
	RETURN;
END_IF

(*to S52_QuickStop*)	
IF NOT nControl.b2_QuickStop THEN
	_eState := E_ProfidriveGSM_State.S52_QuickStop;
	RETURN;
END_IF

(*to S2_ReadyForSwitchingOn*)	
IF NOT nControl.b3_EnableOperation OR bStandstill THEN
	_eState := E_ProfidriveGSM_State.S2_ReadyForSwitchingOn;
END_IF

(*to S4_Operation*)	
IF nControl.b0_On THEN
	_eState := E_ProfidriveGSM_State.S4_Operation;
	RETURN;
END_IF
END_METHOD

{ attribute 'hide' }
METHOD INTERNAL S52_QuickStop
VAR_INPUT
END_VAR
nStatus.b0_ReadyToSwitchOn 		:= TRUE;				
nStatus.b1_ReadyForOperation 	:= TRUE;				
nStatus.b2_OperationEnabled 	:= FALSE;					
nStatus.b6_SwitchingOnInhibited := FALSE;

(*to S1_SwitchingOnInhibited*)	
IF NOT nControl.b1_CoastStop THEN
	_eState := E_ProfidriveGSM_State.S1_SwitchingOnInhibited;
	RETURN;
END_IF

(*to S1_SwitchingOnInhibited*)	
IF NOT nControl.b3_EnableOperation OR bStandstill THEN
	_eState := E_ProfidriveGSM_State.S1_SwitchingOnInhibited;
END_IF
END_METHOD

END_FUNCTION_BLOCK

// Common/ProfidriveParamInterpreter/FB_ProfidriveParamInterpreter
FUNCTION_BLOCK PUBLIC FB_ProfidriveParamInterpreter
VAR_INPUT
	(* Pointer to raw user data *)
	pRawData		: POINTER TO BYTE;
	(* Pointer to array of parameters *)
	pParamSet		: POINTER TO ST_ProfidriveParam_Set;
END_VAR
VAR_OUTPUT
	(* Reference number for response *)
	nReference		: BYTE;
	(* 1 = read, 2 = write *)
	nCommand		: BYTE;
	(* Addressed axis number *)
	nAxis			: BYTE;
	(* Number of parameters to read/write *)
	nParameters		: BYTE;
END_VAR
VAR
	nOffsReq		: BYTE;
	nOffsValue		: BYTE;
	nFormatSize		: BYTE;
	nValues			: BYTE;
	i, j, k			: UINT;
END_VAR

(* Copy header (first 4 bytes) *)
	nReference := pRawData[0];
	nCommand := pRawData[1];
	nAxis := pRawData[2];
	nParameters := pRawData[3];

(* Set request offset behind header *)
	nOffsReq := 4;

(* Set value offset behind last request *)
	nOffsValue := 4 + nParameters * 6;

(* Reset all parameters *)
	memset(pParamSet, 0, SIZEOF(ST_ProfidriveParam_Set));

(* Check parameter number *)	
	IF nParameters = 0 THEN
		RETURN;
	END_IF

(* Loop through number of parameter requests *)
	FOR i := 0 TO nParameters - 1 BY 1 DO
		
		(* Get parameter request information (6 bytes)... *)
		pParamSet^[i].nAttribute := pRawData[nOffsReq];
		pParamSet^[i].nElements := pRawData[nOffsReq + 1];
		pParamSet^[i].nNumber := pRawData[nOffsReq + 2] * 16#100 + pRawData[nOffsReq + 3];
		pParamSet^[i].nSubIndex := pRawData[nOffsReq + 4] * 16#100 + pRawData[nOffsReq + 5];
		
		(* ... and set offset to next request *)
		nOffsReq := nOffsReq + 6;
				
		(* Write command -> get values *)
		IF nCommand = 2 THEN		
			(* Get format *)
			nFormatSize := FormatSize(pRawData[nOffsValue]);
			pParamSet^[i].nFormat := FormatType(pRawData[nOffsValue]);
			nOffsValue := nOffsValue + 1;
			
			(* Get number of values *)
			nValues := pRawData[nOffsValue];
			nOffsValue := nOffsValue + 1;
			
			(* Loop through number of values *)
			FOR j := 0 TO nValues - 1 BY 1 DO
				
				(* Set value offset behind current values *)
				nOffsValue := nOffsValue + nFormatSize;
				
				(* Loop through format size and get values in reverse order *)
				FOR k := 0 TO nFormatSize - 1 BY 1 DO
					pParamSet^[i].aValue[j + k] := pRawData[nOffsValue - k - 1];
				END_FOR
			END_FOR
			
			(* Check if odd and set to even number *)
			IF nOffsValue.0 THEN
				nOffsValue := nOffsValue + 1;
			END_IF
		END_IF
	END_FOR

METHOD INTERNAL FormatSize : BYTE
VAR_INPUT
	nFormat	: BYTE;
END_VAR
CASE nFormat OF
	 16#02 : FormatSize := 2;
	 16#03 : FormatSize := 2;
	 16#04 : FormatSize := 4;
	 16#05 : FormatSize := 2;
	 16#06 : FormatSize := 2;
	 16#07 : FormatSize := 4;
	 16#08 : FormatSize := 4;
	 16#40 : FormatSize := 0;
	 16#41 : FormatSize := 2;
	 16#42 : FormatSize := 2;
	 16#43 : FormatSize := 4;
	 16#44 : FormatSize := 0;
ELSE
	FormatSize := 0;
END_CASE
END_METHOD

METHOD INTERNAL FormatType : E_ProfidriveParam_Format
VAR_INPUT
	nFormat	: BYTE;
END_VAR
CASE nFormat OF
	 16#02 : FormatType := E_ProfidriveParam_Format.INT8;
	 16#03 : FormatType := E_ProfidriveParam_Format.INT16;
	 16#04 : FormatType := E_ProfidriveParam_Format.INT32;
	 16#05 : FormatType := E_ProfidriveParam_Format.UINT8;
	 16#06 : FormatType := E_ProfidriveParam_Format.UINT16;
	 16#07 : FormatType := E_ProfidriveParam_Format.UINT32;
	 16#08 : FormatType := E_ProfidriveParam_Format.FLOAT;
	 16#40 : FormatType := E_ProfidriveParam_Format.ZERO;
	 16#41 : FormatType := E_ProfidriveParam_Format.BYTE_;
	 16#42 : FormatType := E_ProfidriveParam_Format.WORD_;
	 16#43 : FormatType := E_ProfidriveParam_Format.DWORD_;
	 16#44 : FormatType := E_ProfidriveParam_Format.ERROR;
ELSE
	FormatType := E_ProfidriveParam_Format.UNKNOWN;
END_CASE
END_METHOD

METHOD INTERNAL MakeResponse : BOOL
VAR_INPUT
	(* Pointer to acyclic user data *)
	pResData		: POINTER TO BYTE;
END_VAR
VAR
	nOffset			: BYTE;
	nFormatSize		: BYTE;
	i, j, k			: UINT;
END_VAR
(* Copy header (first 4 bytes) *)
	pResData[0] := nReference;
	pResData[1] := nCommand;
	pResData[2] := nAxis;
	pResData[3] := nParameters;

(* Set offset behind header *)
	nOffset := 4;
	
(* Check parameter number *)	
	IF nParameters = 0 THEN
		RETURN;
	END_IF

(* Loop through number of parameter requests *)
	FOR i := 0 TO nParameters - 1 BY 1 DO
		
		(* Set format *)
		pResData[nOffset] := pParamSet^[i].nFormat;
		nFormatSize := FormatSize(pParamSet^[i].nFormat);
		nOffset := nOffset + 1;
		
		(* Set number of values *)
		pResData[nOffset] := pParamSet^[i].nElements;
		nOffset := nOffset + 1;
		
		(* Loop through number of elements *)
		FOR j := 0 TO pParamSet^[i].nElements - 1 BY 1 DO
			
			(* Set value offset behind current values *)
			nOffset := nOffset + nFormatSize;
			
			(* Loop through format size and get values in reverse order *)
			
			IF nFormatSize > 0 THEN
				FOR k := 0 TO nFormatSize - 1 BY 1 DO
					pResData[nOffset - k - 1] := pParamSet^[i].aValue[j + k] ;
				END_FOR
			END_IF
			
		END_FOR
		
		(* Check if odd and set to even number *)
		IF nOffset.0 THEN
			nOffset := nOffset + 1;
		END_IF	
	END_FOR

(* Return true when finished *)
	MakeResponse := TRUE;
END_METHOD

METHOD INTERNAL Reset : BOOL
nReference := 0;
nCommand := 0;
nAxis := 0;
nParameters := 0;
memset(pParamSet, 0, SIZEOF(ST_ProfidriveParam_Set));
END_METHOD

END_FUNCTION_BLOCK

// Common/Utils/F_CalcCrc16
FUNCTION F_CalcCrc16 : WORD
VAR_INPUT
	pData		: POINTER TO BYTE;
	nDataSize	: INT;
	nInitCRC	: WORD;
	nPolynom	: WORD;
END_VAR
VAR
	nCrc		: WORD;
	nDataX		: BYTE;
	nI			: INT;
	nJ			: INT;
END_VAR

nCrc := nInitCRC;

FOR nI := 0 TO nDataSize - 1 BY 1 DO
	nDataX	:= pData[nI];
	FOR nJ := 0 TO 7 BY 1 DO
		IF (SHR(nCrc,15) AND 1) <> (SHR(nDataX,7) AND 1) THEN
			nCrc := SHL(nCrc,1) XOR nPolynom;
		ELSE
			nCrc := SHL(nCrc,1);
		END_IF
		nDataX := SHL(nDataX,1);
	END_FOR	
END_FOR

F_CalcCrc16 := nCrc;

END_FUNCTION

// Devices/Profidrive_Telegram1/FB_Profidrive_Telegram1
{attribute 'reflection'} 
FUNCTION_BLOCK FB_Profidrive_Telegram1 EXTENDS FB_LinkDataReal
VAR_INPUT	
	pControl 			: PVOID; //Pocess data from fieldbus. Size must be >= stControl.
	pStatus 			: PVOID; //Pocess data to fieldbus. Size must be >= stStatus.
	stControl 			: ST_Profidrive_Telegram1_Control; //Control structure. Is read from the fieldbus.
	stConfig 			: ST_Profidrive_Telegram1_Config; //Config structure. Contains parameters of the device.	
END_VAR

VAR_OUTPUT
	stStatus					: ST_Profidrive_Telegram1_Status;
	fValue						: REAL;
END_VAR

VAR
    {attribute 'instance-path'} 
    {attribute 'noinit'} 
    _sPath 						: STRING; 	
	                        	
	_fbProfidriveGSM			: FB_ProfidriveGSM;	
	_fbMoveVelocity				: FB_MoveVelocity;
	                        	
	_fAcceleration	 			: REAL;
	_fDeceleration		 		: REAL;
	_fDecelerationQuickStop 	: REAL;
	_fDecelerationCoastStop 	: REAL;
	_bQuickStopExternal			: BOOL;	
END_VAR

SUPER^();
InitRun();

GetControlData();
Cycle();
SetStatusData();

METHOD INTERNAL Cycle
(*Initialize Init Value*)
IF SUPER^.Status.7 THEN
	ControlData := StatusData;
END_IF

(* Call base statemachine *)
_fbProfidriveGSM.bStandstill					:= OC_Core.F_Compare(_fbMoveVelocity.fVelocity, 0, 1E-3);
_fbProfidriveGSM.nControl.b0_On 				:= stControl.b0_OFF1;
_fbProfidriveGSM.nControl.b1_CoastStop 			:= stControl.b1_OFF2;
_fbProfidriveGSM.nControl.b2_QuickStop 			:= stControl.b2_OFF3 AND NOT _bQuickStopExternal;
_fbProfidriveGSM.nControl.b3_EnableOperation	:= stControl.b3_EnableOperation;

(* Preset target values *)
_fbMoveVelocity.fTargetVelocity					:= 0;
_fbMoveVelocity.fAccMax 						:= _fAcceleration;
_fbMoveVelocity.fDecMax 						:= _fDeceleration;

(* Operation Logic *)
Operation();
	
(* Coast stop, Quick stop, Ramp stop *)
IF _fbProfidriveGSM.eState = E_ProfidriveGSM_State.S1_SwitchingOnInhibited THEN
	_fbMoveVelocity.fTargetVelocity := 0;
	_fbMoveVelocity.fAccMax := _fDecelerationCoastStop;
	_fbMoveVelocity.fDecMax := _fDecelerationCoastStop;
ELSIF _fbProfidriveGSM.eState = E_ProfidriveGSM_State.S52_QuickStop THEN
	_fbMoveVelocity.fTargetVelocity := 0;
	_fbMoveVelocity.fAccMax := _fDecelerationQuickStop;
	_fbMoveVelocity.fDecMax := _fDecelerationQuickStop;
ELSIF _fbProfidriveGSM.eState = E_ProfidriveGSM_State.S51_RampStop THEN
	_fbMoveVelocity.fTargetVelocity := 0;
	_fbMoveVelocity.fAccMax := _fDeceleration;
	_fbMoveVelocity.fDecMax := _fDeceleration;
END_IF

(* Call MoveVelocity *)
_fbMoveVelocity();
	
(* Status word *)
stStatus.b0_ReadyForSwitchingOn				:= _fbProfidriveGSM.nStatus.b0_ReadyToSwitchOn;	
stStatus.b1_ReadyForOperation				:= _fbProfidriveGSM.nStatus.b1_ReadyForOperation;
stStatus.b2_OperationEnabled				:= stControl.b3_EnableOperation;
stStatus.b3_FaultPresent					:= FALSE;
stStatus.b4_NoCoastDownActive				:= _fbProfidriveGSM.eState <> E_ProfidriveGSM_State.S1_SwitchingOnInhibited;
stStatus.b5_NoQuickStopActive				:= _fbProfidriveGSM.eState <> E_ProfidriveGSM_State.S52_QuickStop;
stStatus.b6_SwitchingOnInhibited			:= _fbProfidriveGSM.nStatus.b6_SwitchingOnInhibited;
stStatus.b7_AlarmPresent					:= FALSE;
stStatus.b8_DeviationWithinTolerance		:= TRUE;
stStatus.b9_ControlRequested				:= stConfig.bControlRequested;
stStatus.b10_RpmCompValueReachedOrExceeded	:= _fbMoveVelocity.bIsReached;
stStatus.b11_TorqueOrPowerLimitNotReached	:= TRUE;
stStatus.b12_OpenHoldingBrake 				:= _fbProfidriveGSM.eState > E_ProfidriveGSM_State.S3_SwitchedOn;
stStatus.b13_NoOvertempAlarm				:= TRUE;	
stStatus.b14_MotorRotatesForwards			:= _fbMoveVelocity.fVelocity >= 0;
stStatus.b15_NoAlarmNoOvertempPowerUnit		:= TRUE;

(* Reset quickstop from extern *)
IF stControl.b7_AcknowledgeFaults THEN
	_bQuickStopExternal := FALSE;
END_IF

(* Calculate NIST *)
IF stConfig.fP2000 = 0 THEN
	stStatus.nVelocity	:= 0;
ELSE
	stStatus.nVelocity := REAL_TO_INT((_fbMoveVelocity.fVelocity * 16#4000) / stConfig.fP2000);
END_IF

(* Output of actual value *)	
IF stConfig.bOutputVelocity THEN
	ControlData := _fbMoveVelocity.fVelocity;
ELSE
	ControlData := ControlData + _fbMoveVelocity.fVelocity *  GVL_Core.fbSystem.fDeltaTime * GVL_Core.fbSystem.fTimeScaling;
END_IF

fValue := ControlData;
END_METHOD

METHOD INTERNAL GetControlData : BOOL
IF pControl <= 0 OR stConfig.bForceMode THEN RETURN; END_IF

F_Memcpy(ADR(stControl), pControl, 2, stConfig.bSwapProcessData);
F_Memcpy(ADR(stControl) + 2, pControl + 2, 2, stConfig.bSwapProcessData);
END_METHOD

METHOD INTERNAL InitRun : BOOL
VAR_INST
	bInitRun : BOOL := TRUE;
END_VAR
IF NOT bInitRun THEN RETURN; END_IF
bInitRun := FALSE;

IF pControl = 0 OR pStatus = 0 THEN
	ADSLOGSTR(ADSLOG_MSGTYPE_WARN, CONCAT(_sPath, ': %s'), 'Plc address not set.');
END_IF
END_METHOD

METHOD PRIVATE Operation : BOOL
IF _fbProfidriveGSM.eState = E_ProfidriveGSM_State.S4_Operation THEN	
	// Main setpoint
	IF NOT stControl.b8_Jog1 AND NOT stControl.b9_Jog2 THEN
		_fbMoveVelocity.fTargetVelocity := (stControl.nTargetVelocity * stConfig.fP2000) / 16#4000;
	// Jog 1
	ELSIF stControl.b8_Jog1 AND NOT stControl.b9_Jog2 THEN
		_fbMoveVelocity.fTargetVelocity := stConfig.fP1058;
	// Jog 2
	ELSIF NOT stControl.b8_Jog1 AND stControl.b9_Jog2 THEN	
		_fbMoveVelocity.fTargetVelocity := stConfig.fP1059;
	END_IF
	// Stop
	IF NOT stControl.b4_OperatingCondition OR NOT stControl.b6_EnableSetpoint THEN
		_fbMoveVelocity.fTargetVelocity := 0;
	END_IF
	// Invert velocity
	IF stControl.b11_SetpointInversion THEN
		_fbMoveVelocity.fTargetVelocity := -_fbMoveVelocity.fTargetVelocity;
	END_IF	
	// Hold velocity
	IF NOT stControl.b5_ContinueRampFunctionGenerator AND NOT stControl.b8_Jog1 AND NOT stControl.b9_Jog2 THEN
		_fbMoveVelocity.fTargetVelocity := _fbMoveVelocity.fVelocity;
	END_IF	
END_IF
END_METHOD

METHOD INTERNAL SetStatusData
IF pStatus <= 0 THEN RETURN; END_IF

F_Memcpy(pStatus, ADR(stStatus), 2, stConfig.bSwapProcessData);
F_Memcpy(pStatus + 2, ADR(stStatus) + 2, 2, stConfig.bSwapProcessData);
END_METHOD

END_FUNCTION_BLOCK

// Devices/SEW_MoviC_Position/FB_SEW_MoviC_Position
(*
FB_SEW_MoviC_Position simulates the funcitionalty of a SEW‑EURODRIVE MOVI-C® CONTROLLER with MOVIKIT® Positioning module.

Disclaimer: This simulation is an independent project and is not affiliated with, endorsed by, or approved by SEW‑EURODRIVE. All rights to the SEW‑EURODRIVE brand name and trademarks remain the property of the manufacturer.
Furthermore, no guarantee is given for the completeness of the functional scope or the error-free operation of the simulation. Users should be aware that deviations from the actual product may occur.
*)

{attribute 'reflection'}
FUNCTION_BLOCK FB_SEW_MoviC_Position EXTENDS FB_LinkDataReal
VAR_INPUT
	pControl 			: PVOID; //Pocess data from fieldbus. Size must be >= stControl.
	pStatus 			: PVOID; //Pocess data to fieldbus. Size must be >= stStatus.
	stControl 			: ST_SEW_MoviC_Position_Control; //Control structure. Is read from the fieldbus.
	stConfig 			: ST_SEW_MoviC_Position_Config; //Config structure. Contains parameters of the device.		
	
	bSTO				: BOOL := TRUE;
	iMovisafe			: I_SEW_Movisafe;	
	nDigitalInputs		: WORD;
END_VAR

VAR_OUTPUT
	stStatus			: ST_SEW_MoviC_Position_Status;
	fValue				: REAL;
END_VAR

VAR
    {attribute 'instance-path'} 
    {attribute 'noinit'} 
    _sPath 				: STRING;	                			
	                			
	_fbBaseState		: FB_ProfidriveGSM;
	_fbBasicDrive		: FB_DriveControl;
	                				
	_bOpModeValid		: BOOL;
END_VAR

SUPER^();
InitRun();

GetControlData();
Safety();
Cycle();
SetStatusData();

METHOD INTERNAL Cycle
//Unity Init - Load persistent data
IF SUPER^.Status.7 THEN
	IF stConfig.fRatioPosition <> 0 THEN	
		_fbBasicDrive.fPosition := SUPER^.StatusData/stConfig.fRatioPosition - stConfig.fPositionOffset;
	ELSE
		_fbBasicDrive.fPosition := SUPER^.StatusData - stConfig.fPositionOffset;
	END_IF
END_IF

(* Evaluate incoming operation mode *)
_bOpModeValid := FALSE;

CASE stControl.nTargetApplicationMode OF
	E_SEW_MoviC_Position_OperationMode.Jog:
		_bOpModeValid := TRUE;
	E_SEW_MoviC_Position_OperationMode.JogNoEnc:
		_bOpModeValid := TRUE;
	E_SEW_MoviC_Position_OperationMode.SpeedControl:
		_bOpModeValid := TRUE;
	E_SEW_MoviC_Position_OperationMode.ReferenceParam:
		_bOpModeValid := TRUE;
	E_SEW_MoviC_Position_OperationMode.ReferenceBus:
		_bOpModeValid := TRUE;
	E_SEW_MoviC_Position_OperationMode.PositionAbs, E_SEW_MoviC_Position_OperationMode.EnergyOptimized, E_SEW_MoviC_Position_OperationMode.MechanicsOptimized:
		_bOpModeValid := TRUE;
	E_SEW_MoviC_Position_OperationMode.PositionRel:
		_bOpModeValid := TRUE;
	E_SEW_MoviC_Position_OperationMode.PositionModPos:
		_bOpModeValid := TRUE;
	E_SEW_MoviC_Position_OperationMode.PositionModNeg:
		_bOpModeValid := TRUE;
	E_SEW_MoviC_Position_OperationMode.PositionModShort:
		_bOpModeValid := TRUE;
END_CASE

(* Base state of the controller *)
_fbBaseState.bStandstill := OC_Core.F_Compare(_fbBasicDrive.fVelocity, 0, 1E-3);
_fbBaseState.nControl.b0_On := stControl.b1_EnableBusStop AND _fbBaseState.eState <> E_ProfidriveGSM_State.S1_SwitchingOnInhibited;
_fbBaseState.nControl.b1_CoastStop := NOT stControl.b13_ActivateInhibit AND bSTO;
_fbBaseState.nControl.b2_QuickStop := stControl.b0_EnableEStop;
_fbBaseState.nControl.b3_EnableOperation := stControl.b7_StartStop AND _bOpModeValid;

_fbBaseState();
		
(* Set parameter of basic drive *)
IF stControl.b12_DisableSoftwareLimits THEN
	_fbBasicDrive.fPositionLimitMin := -2147483648.0;
	_fbBasicDrive.fPositionLimitMax := 2147483647.0;
	_fbBasicDrive.fTolerance := 0.1;
ELSE
	_fbBasicDrive.fPositionLimitMin := DINT_TO_REAL(stConfig.nSoftwareLimitMin);
	_fbBasicDrive.fPositionLimitMax := DINT_TO_REAL(stConfig.nSoftwareLimitMax);
	_fbBasicDrive.fTolerance := 0.1;
END_IF
					
(* Evaluate base state *)
CASE _fbBaseState.eState OF
	
(* S1, S2 or S3 -> Drive coasts to a stop or brake is applied *)
	E_ProfidriveGSM_State.S1_SwitchingOnInhibited,
	E_ProfidriveGSM_State.S2_ReadyForSwitchingOn,
	E_ProfidriveGSM_State.S3_SwitchedOn:
		_fbBasicDrive.Stop(stConfig.fDecCoastStop);

(* S4 -> Evaluate operation mode *)
	E_ProfidriveGSM_State.S4_Operation:
		Operation();

(* S5a -> Drive decelerates with application limit *)
	E_ProfidriveGSM_State.S51_RampStop:
		_fbBasicDrive.Stop(stConfig.fDecelerationLimit);
		
(* S5b -> Drive decelerates with emergency stop ramp *)
	E_ProfidriveGSM_State.S52_QuickStop:
	    _fbBasicDrive.Stop(stConfig.fDecEstop);
END_CASE
	
(* Status Word *)
stStatus.b0_InverterReady				:= TRUE;
stStatus.b1_STOInactive					:= bSTO;
stStatus.b2_PowerStageOn				:= stControl.b13_ActivateInhibit;
stStatus.b3_BrakeReleased				:= stControl.b1_EnableBusStop OR stControl.b3_ReleaseBrake;
stStatus.b4_MotorTurning				:= NOT _fbBaseState.bStandstill;
stStatus.b5_DriveReferenced				:= TRUE;
stStatus.b6_SetpointsActive		 		:= FALSE;
stStatus.b7_TargetpositionReached		:= _fbBasicDrive.bIsPositionReached;	
stStatus.b8_ErrorActive					:= FALSE;
stStatus.b9_WarningActive				:= FALSE;
stStatus.b10_DriveTrain2Active			:= stControl.b10_ActivateDriveTrain2;
stStatus.b11_SpeedSetpointReached		:= _fbBasicDrive.bIsMoving;
stStatus.b12_SoftwareLimitsDisabled		:= stControl.b12_DisableSoftwareLimits;
stStatus.b13_OutputStageInhibit			:= _fbBaseState.nStatus.b6_SwitchingOnInhibited;
stStatus.b14_StandByModeActive			:= stControl.b14_ActivateStandByMode;
stStatus.b15_MovikitHeartbeat			:= stControl.b15_MovikitHeartbeat;

(* Status values *)
stStatus.nActualSpeed := REAL_TO_INT(_fbBasicDrive.fVelocity / stConfig.fRatioVelocity);
stStatus.nActualStatus := 0;
stStatus.nActualTorque := 0;
stStatus.nDigitalInputs := nDigitalInputs;
IF _bOpModeValid THEN
	stStatus.nActualApplicationMode := stControl.nTargetApplicationMode;
END_IF
stStatus.nActualPosition := REAL_TO_DINT(_fbBasicDrive.fPosition);
	
(* Position output *)
THIS^.ControlData := _fbBasicDrive.fPosition * stConfig.fRatioPosition + stConfig.fPositionOffset;
fValue := ControlData;
END_METHOD

METHOD INTERNAL GetControlData : BOOL
IF pControl <= 0 OR stConfig.bForceMode THEN RETURN; END_IF

(* PO1 Control Word *)
F_Memcpy(ADR(stControl), pControl, 2, stConfig.bSwapProcessData);
(* PO2 Setpoint Speed *)
F_Memcpy(ADR(stControl) + 2, pControl + 2, 2, stConfig.bSwapProcessData);
(* PO3 Setpoint Acceleration *)
F_Memcpy(ADR(stControl) + 4, pControl + 4, 2, stConfig.bSwapProcessData);
(* PO4 Setpoint Deceleration *)
F_Memcpy(ADR(stControl) + 6, pControl + 6, 2, stConfig.bSwapProcessData);
(* PO5 Digital Outputs *)
F_Memcpy(ADR(stControl) + 8, pControl + 8, 2, stConfig.bSwapProcessData);
(* PO6 Target Application Mode *)
F_Memcpy(ADR(stControl) + 10, pControl + 10, 2, stConfig.bSwapProcessData);
(* PO7,PO8 Target Position *)
F_Memcpy(ADR(stControl) + 12, pControl + 12, 4, stConfig.bSwapProcessData);
END_METHOD

METHOD INTERNAL InitRun
VAR_INST
	bInitRun : BOOL := TRUE;
END_VAR
IF NOT bInitRun THEN RETURN; END_IF
bInitRun := FALSE;

IF pControl = 0 OR pStatus = 0 THEN
	ADSLOGSTR(ADSLOG_MSGTYPE_WARN, CONCAT(_sPath, ': %s'), 'Plc address not set.');
END_IF

_fbBasicDrive.fPosition := stConfig.fInitPosition;
END_METHOD

METHOD PRIVATE Operation
VAR_INST
	fTargetPos			: REAL;
	fSetpointVel		: REAL;
	fSetpointAcc		: REAL;
	fSetpointDec		: REAL;
END_VAR
(* Copy setpoint values *)
fTargetPos 		:= DINT_TO_REAL(stControl.nTargetPosition);
fSetpointVel 	:= stControl.nSetpointSpeed * stConfig.fRatioVelocity; 
fSetpointAcc 	:= stControl.nSetpointAcceleration * stConfig.fRatioAccDec;
fSetpointDec 	:= stControl.nSetpointDeceleration * stConfig.fRatioAccDec;

(* Operation statemachine *)
CASE stStatus.nActualApplicationMode OF	
	E_SEW_MoviC_Position_OperationMode.Jog:
		IF stControl.b4_JoggingCW AND NOT stControl.b5_JoggingCCW THEN
			_fbBasicDrive.MoveAbsolute(DINT_TO_REAL(stConfig.nSoftwareLimitMax), fSetpointVel, fSetpointAcc, fSetpointDec);
		ELSIF stControl.b5_JoggingCCW AND NOT stControl.b4_JoggingCW THEN
			_fbBasicDrive.MoveAbsolute(DINT_TO_REAL(stConfig.nSoftwareLimitMin), fSetpointVel, fSetpointAcc, fSetpointDec);
		ELSE
			_fbBasicDrive.Stop(fSetpointDec);
		END_IF
		
	E_SEW_MoviC_Position_OperationMode.JogNoEnc:			
		IF stControl.b4_JoggingCW AND NOT stControl.b5_JoggingCCW THEN
			_fbBasicDrive.MoveVelocity(fSetpointVel, fSetpointAcc, fSetpointDec);
		ELSIF stControl.b5_JoggingCCW AND NOT stControl.b4_JoggingCW THEN
			_fbBasicDrive.MoveVelocity(-fSetpointVel, fSetpointAcc, fSetpointDec);
		ELSE
			_fbBasicDrive.Stop(fSetpointDec);
		END_IF
		
	E_SEW_MoviC_Position_OperationMode.SpeedControl:
		_fbBasicDrive.MoveVelocity(fSetpointVel, fSetpointAcc, fSetpointDec);
	
	E_SEW_MoviC_Position_OperationMode.ReferenceParam:
		//not yet implemented
		
	E_SEW_MoviC_Position_OperationMode.ReferenceBus:
		//not yet implemented
	
	E_SEW_MoviC_Position_OperationMode.PositionAbs, E_SEW_MoviC_Position_OperationMode.EnergyOptimized, E_SEW_MoviC_Position_OperationMode.MechanicsOptimized:
		IF stControl.b7_StartStop THEN						
			_fbBasicDrive.MoveAbsolute(fTargetPos, fSetpointVel, fSetpointAcc, fSetpointDec);
		ELSE
			_fbBasicDrive.Stop(fSetpointDec);
		END_IF
	
	E_SEW_MoviC_Position_OperationMode.PositionRel:
		//not yet implemented
		
	E_SEW_MoviC_Position_OperationMode.PositionModPos:
		//not yet implemented
		
	E_SEW_MoviC_Position_OperationMode.PositionModNeg:
		//not yet implemented
		
	E_SEW_MoviC_Position_OperationMode.PositionModShort:
		//not yet implemented
END_CASE
END_METHOD

METHOD INTERNAL Safety
VAR_INPUT
END_VAR
(* Check if Movisafe is available *)
IF iMovisafe <> 0 THEN
	bSTO := iMovisafe.bSTO;
END_IF
END_METHOD

METHOD INTERNAL SetStatusData
IF pStatus <= 0 THEN RETURN; END_IF

(* PI1 Status Word *)
F_Memcpy(pStatus, ADR(stStatus), 2, stConfig.bSwapProcessData);
(* PI2 Actual Speed *)
F_Memcpy(pStatus + 2, ADR(stStatus) + 2, 2, stConfig.bSwapProcessData);
(* PI3 Actual Status *)
F_Memcpy(pStatus + 4, ADR(stStatus) + 4, 2, stConfig.bSwapProcessData);
(* PI4 Actual Torque *)
F_Memcpy(pStatus + 6, ADR(stStatus) + 6, 2, stConfig.bSwapProcessData);
(* PI5 Digital Inputs *)
F_Memcpy(pStatus + 8, ADR(stStatus) + 8, 2, stConfig.bSwapProcessData);
(* PI6 Actual Application Mode *)
F_Memcpy(pStatus + 10, ADR(stStatus) + 10, 2, stConfig.bSwapProcessData);
(* PI7,PI8 Actual Position *)
F_Memcpy(pStatus + 12, ADR(stStatus) + 12, 4, stConfig.bSwapProcessData);
END_METHOD

END_FUNCTION_BLOCK

// Devices/I_SEW_Movisafe
INTERFACE I_SEW_Movisafe

PROPERTY bSTO : BOOL
GET
END_GET
END_PROPERTY

END_INTERFACE

// Devices/SEW_MoviC_Velocity/FB_SEW_MoviC_Velocity
(*
FB_SEW_MoviC_Velocity simulates the funcitionalty of a SEW‑EURODRIVE MOVI-C® CONTROLLER with MOVIKIT® Velocity module.

Disclaimer: This simulation is an independent project and is not affiliated with, endorsed by, or approved by SEW‑EURODRIVE. All rights to the SEW‑EURODRIVE brand name and trademarks remain the property of the manufacturer.
Furthermore, no guarantee is given for the completeness of the functional scope or the error-free operation of the simulation. Users should be aware that deviations from the actual product may occur.
*)

{attribute 'reflection'}
FUNCTION_BLOCK FB_SEW_MoviC_Velocity EXTENDS FB_LinkDataReal

VAR_INPUT
	pControl 			: PVOID; //Pocess data from fieldbus. Size must be >= stControl.
	pStatus 			: PVOID; //Pocess data to fieldbus. Size must be >= stStatus.
	stControl 			: ST_SEW_MoviC_Velocity_Control; //Control structure. Is read from the fieldbus.
	stConfig 			: ST_SEW_MoviC_Velocity_Config; //Config structure. Contains parameters of the device.	
	
	bSTO				: BOOL := TRUE;
	iMovisafe			: I_SEW_Movisafe;
END_VAR

VAR_OUTPUT
	stStatus			: ST_SEW_MoviC_Velocity_Status;
	fValue				: REAL;
END_VAR

VAR
    {attribute 'instance-path'} 
    {attribute 'noinit'} 
    _sPath 				: STRING; 	                			
	                			
	_fbBaseState		: FB_ProfidriveGSM;
	_fbBasicDrive		: FB_DriveControl;	                						
END_VAR

SUPER^();
InitRun();

GetControlData();
Safety();
Cycle();
SetStatusData();

METHOD INTERNAL Cycle
(* Base state of the controller *)
_fbBaseState.bStandstill := OC_Core.F_Compare(_fbBasicDrive.fVelocity, 0, 1E-3);
_fbBaseState.nControl.b0_On := stControl.b1_EnableBusStop AND _fbBaseState.eState <> E_ProfidriveGSM_State.S1_SwitchingOnInhibited;
_fbBaseState.nControl.b1_CoastStop := NOT stControl.b13_ActivateInhibit AND bSTO;
_fbBaseState.nControl.b2_QuickStop := stControl.b0_EnableEStop;
_fbBaseState.nControl.b3_EnableOperation := stControl.b7_StartStop;

_fbBaseState();
					
(* Evaluate base state *)
CASE _fbBaseState.eState OF	
(* S1, S2 or S3 -> Drive coasts to a stop or brake is applied *)
	E_ProfidriveGSM_State.S1_SwitchingOnInhibited,
	E_ProfidriveGSM_State.S2_ReadyForSwitchingOn,
	E_ProfidriveGSM_State.S3_SwitchedOn:
		_fbBasicDrive.Stop(stConfig.fDecCoastStop);

(* S4 -> Operation mode *)
	E_ProfidriveGSM_State.S4_Operation:
		Operation();

(* S5a -> Drive decelerates with application limit *)
	E_ProfidriveGSM_State.S51_RampStop:
		_fbBasicDrive.Stop(stConfig.fDecelerationLimit);
		
(* S5b -> Drive decelerates with emergency stop ramp *)
	E_ProfidriveGSM_State.S52_QuickStop:
	    _fbBasicDrive.Stop(stConfig.fDecEstop);
END_CASE
	
(* Status Word *)
stStatus.b0_InverterReady				:= TRUE;
stStatus.b1_STOInactive					:= bSTO;
stStatus.b2_PowerStageOn				:= _fbBaseState.bPowerOn;
stStatus.b3_BrakeReleased				:= stControl.b1_EnableBusStop OR stControl.b3_ReleaseBrake;
stStatus.b4_MotorTurning				:= NOT _fbBaseState.bStandstill;
stStatus.b5_DriveReferenced				:= TRUE;
stStatus.b6_SetpointsActive		 		:= FALSE;
stStatus.b7_TargetpositionReached		:= FALSE;	
stStatus.b8_ErrorActive					:= FALSE;
stStatus.b9_WarningActive				:= FALSE;
stStatus.b10_DriveTrain2Active			:= stControl.b10_ActivateDriveTrain2;
stStatus.b11_SpeedSetpointReached		:= _fbBasicDrive.bIsMoving;
stStatus.b12_SoftwareLimitsDisabled		:= stControl.b12_DisableSoftwareLimits;
stStatus.b13_OutputStageInhibit			:= _fbBaseState.nStatus.b6_SwitchingOnInhibited;
stStatus.b14_StandByModeActive			:= stControl.b14_ActivateStandByMode;
stStatus.b15_MovikitHeartbeat			:= stControl.b15_MovikitHeartbeat;

(* Status values *)
stStatus.nActualSpeed := REAL_TO_INT(_fbBasicDrive.fVelocity / stConfig.fRatioVelocity);
stStatus.nActualStatus := 0;
stStatus.nActualTorque := 0;
stStatus.nDigitalInputs := 0;
	
(* Output of actual value *)	
IF stConfig.bOutputVelocity THEN
	ControlData := _fbBasicDrive.fVelocity / stConfig.fRatioVelocity;
ELSE
	ControlData := ControlData + _fbBasicDrive.fVelocity / stConfig.fRatioVelocity *  GVL_Core.fbSystem.fDeltaTime * GVL_Core.fbSystem.fTimeScaling;
END_IF

fValue := ControlData;
END_METHOD

METHOD INTERNAL GetControlData : BOOL
IF pControl <= 0 OR stConfig.bForceMode THEN RETURN; END_IF

(* PO1 Control Word *)
F_Memcpy(ADR(stControl), pControl, 2, stConfig.bSwapProcessData);
(* PO2 Setpoint Speed *)
F_Memcpy(ADR(stControl) + 2, pControl + 2, 2, stConfig.bSwapProcessData);
(* PO3 Setpoint Acceleration *)
F_Memcpy(ADR(stControl) + 4, pControl + 4, 2, stConfig.bSwapProcessData);
(* PO4 Setpoint Deceleration *)
F_Memcpy(ADR(stControl) + 6, pControl + 6, 2, stConfig.bSwapProcessData);
(* PO5 Digital Outputs *)
F_Memcpy(ADR(stControl) + 8, pControl + 8, 2, stConfig.bSwapProcessData);
END_METHOD

METHOD INTERNAL InitRun
VAR_INST
	bInitRun : BOOL := TRUE;
END_VAR
IF NOT bInitRun THEN RETURN; END_IF
bInitRun := FALSE;

IF pControl = 0 OR pStatus = 0 THEN
	ADSLOGSTR(ADSLOG_MSGTYPE_WARN, CONCAT(_sPath, ': %s'), 'Plc address not set.');
END_IF

_fbBasicDrive.fPosition := stConfig.fInitPosition;
END_METHOD

METHOD PRIVATE Operation
VAR_INST
	fTargetPos			: REAL;
	fSetpointVel		: REAL;
	fSetpointAcc		: REAL;
	fSetpointDec		: REAL;
END_VAR
(* Copy setpoint values *)
fSetpointVel 	:= stControl.nSetpointSpeed * stConfig.fRatioVelocity; 
fSetpointAcc 	:= stControl.nSetpointAcceleration * stConfig.fRatioAccDec;

_fbBasicDrive.MoveVelocity(fSetpointVel, fSetpointAcc, fSetpointAcc);
END_METHOD

METHOD INTERNAL Safety
VAR_INPUT
END_VAR
(* Check if Movisafe is available *)
IF iMovisafe <> 0 THEN
	bSTO := iMovisafe.bSTO;
END_IF
END_METHOD

METHOD INTERNAL SetStatusData
IF pStatus <= 0 THEN RETURN; END_IF

(* PI1 Status Word *)
F_Memcpy(pStatus, ADR(stStatus), 2, stConfig.bSwapProcessData);
(* PI2 Actual Speed *)
F_Memcpy(pStatus + 2, ADR(stStatus) + 2, 2, stConfig.bSwapProcessData);
(* PI3 Actual Status *)
F_Memcpy(pStatus + 4, ADR(stStatus) + 4, 2, stConfig.bSwapProcessData);
(* PI4 Actual Torque *)
F_Memcpy(pStatus + 6, ADR(stStatus) + 6, 2, stConfig.bSwapProcessData);
(* PI5 Digital Inputs *)
F_Memcpy(pStatus + 8, ADR(stStatus) + 8, 2, stConfig.bSwapProcessData);
END_METHOD

END_FUNCTION_BLOCK

// Devices/SEW_Movisafe_CSSx1a/FB_SEW_Movisafe_CSSx1a
(*
FB_SEW_Movisafe_CSSx1a simulates the funcitionalty of a SEW‑EURODRIVE MOVISAFE® module.

Disclaimer: This simulation is an independent project and is not affiliated with, endorsed by, or approved by SEW‑EURODRIVE. All rights to the SEW‑EURODRIVE brand name and trademarks remain the property of the manufacturer.
Furthermore, no guarantee is given for the completeness of the functional scope or the error-free operation of the simulation. Users should be aware that deviations from the actual product may occur.
*)

{attribute 'reflection'}
FUNCTION_BLOCK FB_SEW_Movisafe_CSSx1a EXTENDS FB_Base IMPLEMENTS I_SEW_Movisafe
VAR_INPUT
	pControl 			: PVOID; //Pocess data from fieldbus. Size must be >= stControl.
	pStatus 			: PVOID; //Pocess data to fieldbus. Size must be >= stStatus.
	stControl 			: ST_SEW_Movisafe_CSSx1a_Control; //Control structure. Is read from the fieldbus.
	stConfig 			: ST_SEW_Movisafe_CSSx1a_Config; //Config structure. Contains parameters of the device.
	
	bASFDiag			: BOOL; //At least one drive safety function has exceeded a limit
	bSBTActive 			: BOOL; //Brake test is active
	bF_DI0				: BOOL; //State digital input 1
	bF_DI1				: BOOL; //State digital input 2
	bF_DI2				: BOOL; //State digital input 3
	bF_DI3				: BOOL; //State digital input 4
	bSSM1				: BOOL; //SSM 1 ist activated (Safe speed monitoring)
	bSSM2				: BOOL; //SSM 2 ist activated (Safe speed monitoring)
	bSSM3				: BOOL;	//SSM 3 ist activated (Safe speed monitoring)
	bSSM4				: BOOL; //SSM 4 ist activated (Safe speed monitoring)
END_VAR

VAR_OUTPUT	
	stStatus			: ST_SEW_Movisafe_CSSx1a_Status;
END_VAR

VAR
    {attribute 'instance-path'} 
    {attribute 'noinit'} 
    _sPath 				: STRING; 
END_VAR

SUPER^();
InitRun();

GetControlData();
Cycle();
SetStatusData();

PROPERTY bSTO : BOOL
GET
bSTO := stStatus.b0_0_StoActive;
END_GET
END_PROPERTY

METHOD Internal Cycle : BOOL
VAR_INPUT
END_VAR
stStatus.b0_0_STOActive			:= stControl.b0_0_STO;
stStatus.b0_1_ASFDiag			:= bASFDiag;
stStatus.b0_2_SBTActive			:= bSBTActive;
stStatus.b0_3_InputDataValid	:= TRUE;
stStatus.b0_4_MutingEncErr		:= stControl.b0_4_MutingEncErr;
stStatus.b0_5_TestModeActive	:= stControl.b0_5_TestModeActice;
stStatus.b0_6_Warning			:= FALSE;
stStatus.b0_7_ErrorState		:= FALSE;
stStatus.b1_0_F_DI0				:= bF_DI0;
stStatus.b1_1_F_DI1				:= bF_DI1;
stStatus.b1_2_F_DI2				:= bF_DI2;
stStatus.b1_3_F_DI3				:= bF_DI3;
stStatus.b1_4_Reserved			:= FALSE;
stStatus.b1_5_Reserved			:= FALSE;
stStatus.b1_6_Reserved			:= FALSE;
stStatus.b1_7_Reserved			:= FALSE;
stStatus.b2_0_SOS1				:= NOT stControl.b2_0_SOS1;
stStatus.b2_1_Reserved			:= FALSE;
stStatus.b2_2_SSx1				:= NOT stControl.b2_2_SSx1;
stStatus.b2_3_SSx2				:= NOT stControl.b2_3_SSx2;
stStatus.b2_4_SDI1				:= NOT stControl.b2_4_SDI1;
stStatus.b2_5_SDI2				:= NOT stControl.b2_5_SDI2;
stStatus.b2_6_SLI1				:= NOT stControl.b2_6_SLI1;
stStatus.b2_7_SLI2				:= NOT stControl.b2_7_SLI2;
stStatus.b3_0_SLS1				:= NOT stControl.b3_0_SLS1;
stStatus.b3_1_SLS2				:= NOT stControl.b3_1_SLS2;
stStatus.b3_2_SLS3				:= NOT stControl.b3_2_SLS3;
stStatus.b3_3_SLS4				:= NOT stControl.b3_3_SLS4;
stStatus.b3_4_SSR1				:= NOT stControl.b3_4_SSR1;
stStatus.b3_5_SSR2				:= NOT stControl.b3_5_SSR2;
stStatus.b3_6_Reserved			:= FALSE;
stStatus.b3_7_Reserved			:= FALSE;
stStatus.b4_0_SLA1				:= NOT stControl.b4_0_SLA1;
stStatus.b4_1_SLA2				:= NOT stControl.b4_1_SLA2;
stStatus.b4_2_SSM1				:= bSSM1;
stStatus.b4_3_SSM2				:= bSSM2;
stStatus.b4_4_SSM3				:= bSSM3;
stStatus.b4_5_SSM4				:= bSSM4;
stStatus.b4_6_Reserved			:= FALSE;
stStatus.b4_7_Reserved			:= FALSE;
stStatus.b5_0_Reserved			:= FALSE;
stStatus.b5_1_Reserved			:= FALSE;
stStatus.b5_2_Reserved			:= FALSE;
stStatus.b5_3_Reserved			:= FALSE;
stStatus.b5_4_Reserved			:= FALSE;
stStatus.b5_5_Reserved			:= FALSE;
stStatus.b5_6_Reserved			:= FALSE;
stStatus.b5_7_Reserved			:= FALSE;
END_METHOD

METHOD INTERNAL GetControlData
VAR_INPUT
END_VAR
IF pControl <= 0 OR stConfig.bForceMode THEN RETURN; END_IF

F_MEMCPY(ADR(stControl), pControl, SIZEOF(stControl), stConfig.bSwapProcessData);
END_METHOD

METHOD INTERNAL InitRun
VAR_INST
	bInitRun : BOOL := TRUE;
END_VAR
IF NOT bInitRun THEN RETURN; END_IF
bInitRun := FALSE;

IF pControl = 0 OR pStatus = 0 THEN
	ADSLOGSTR(ADSLOG_MSGTYPE_WARN, CONCAT(_sPath, ': %s'), 'Plc address not set.');
END_IF
END_METHOD

METHOD INTERNAL SetStatusData
VAR_INPUT
END_VAR
IF pStatus <= 0 THEN RETURN; END_IF

F_MEMCPY(pStatus, ADR(stStatus), SIZEOF(stStatus), stConfig.bSwapProcessData);
END_METHOD

END_FUNCTION_BLOCK

// Devices/Siemens_RcvDp/FB_Siemens_RcvDp
(*
FB_Siemens_RcvDp simulates the funcitionalty of a Siemens PN/PN coupler RCVDP safety-related communication.

Disclaimer: This simulation is an independent project and is not affiliated with, endorsed by, or approved by Siemens. All rights to the Siemens brand name and trademarks remain the property of the manufacturer.
Furthermore, no guarantee is given for the completeness of the functional scope or the error-free operation of the simulation. Users should be aware that deviations from the actual product may occur.
*)

{attribute 'reflection'} 
FUNCTION_BLOCK FB_Siemens_RcvDp EXTENDS FB_Base
VAR_INPUT
	pControl 			: PVOID; //Pocess data from fieldbus. Size must be >= stControl.
	pStatus 			: PVOID; //Pocess data to fieldbus. Size must be >= stStatus.
	stControl			: ST_Siemens_RcvDp_Control; 
	stConfig 			: ST_Siemens_RcvDp_Config;
	
	stDevData			: ST_Siemens_RcvDp_DevData;
END_VAR

VAR_OUTPUT
	stStatus			: ST_Siemens_RcvDp_Status; 
	
	stHstData			: ST_Siemens_RcvDp_HstData;
END_VAR

VAR
    {attribute 'instance-path'} 
    {attribute 'noinit'} 
    _sPath 				: STRING; 

	_nLastSequenceNumber: WORD;
	_nCalculatedCrc		: WORD;	
	_TonTimeout			: TON;	
END_VAR

VAR CONSTANT
	N_POLYNOM			: WORD := 16#4EAB;
END_VAR

SUPER^();
InitRun();	
GetControlData();
Cycle();
SetStatusData();

METHOD PRIVATE Cycle
VAR_INPUT
END_VAR
(* Simplified communication when using PLCSIM Adv. *)
	IF OC_Core.GVL_Core.fbSystem.eControllerType = E_ControllerType.PlcSimAdvanced THEN
		SimLogic();
		RETURN;
	END_IF

(* Calculate received crc *)
	_nCalculatedCrc := F_CalcCrc16(ADR(stControl), 8, stConfig.nDpDpId, N_POLYNOM);

(* Restart timer, if sequence number has changed *)
	IF stControl.nRcvSequenceNumber <> _nLastSequenceNumber AND NOT stHstData.bError THEN
		_nLastSequenceNumber := stControl.nRcvSequenceNumber;
		stHstData.bSubsOn	:= FALSE;
		_TonTimeout.IN		:= FALSE;
	ELSE
		_TonTimeout.IN		:= TRUE;
	END_IF

(* Reintegration *)
	IF (stConfig.bAutoAckRei AND stHstData.bError) OR stDevData.bAckRei THEN
		stHstData.bError 	:= FALSE;
		_TonTimeout.IN		:= FALSE;
	END_IF

(* Check if timer has expired *)
	_TonTimeout();
	
	IF _TonTimeout.Q	THEN
		stHstData.bError	:= TRUE;
		stHstData.bSubsOn	:= TRUE;
	END_IF

(* compare received crc value with calculated crc *)
	IF stControl.nRcvCrc = _nCalculatedCrc AND NOT stHstData.bError THEN
		stHstData.bSubsOn	:= FALSE;
	ELSE
		stHstData.bError	:= TRUE;
		stHstData.bSubsOn	:= TRUE;
	END_IF

(* Get substitude or safety values *)
	IF stHstData.bSubsOn THEN
		stHstData.bRcv00	:= stDevData.bSub00;
		stHstData.bRcv01	:= stDevData.bSub01;
		stHstData.bRcv02	:= stDevData.bSub02;
		stHstData.bRcv03	:= stDevData.bSub03;
		stHstData.bRcv04	:= stDevData.bSub04;
		stHstData.bRcv05	:= stDevData.bSub05;
		stHstData.bRcv06	:= stDevData.bSub06;
		stHstData.bRcv07	:= stDevData.bSub07;
		stHstData.bRcv08	:= stDevData.bSub08;
		stHstData.bRcv09	:= stDevData.bSub09;
		stHstData.bRcv10	:= stDevData.bSub10;
		stHstData.bRcv11	:= stDevData.bSub11;
		stHstData.bRcv12	:= stDevData.bSub12;
		stHstData.bRcv13	:= stDevData.bSub13;
		stHstData.bRcv14	:= stDevData.bSub14;
		stHstData.bRcv15	:= stDevData.bSub15;
		stHstData.nRcv00	:= stDevData.nSub00;
		stHstData.nRcv01	:= stDevData.nSub01;
	ELSE
		stHstData.bRcv00	:= stControl.nRcvBoolData.0;
		stHstData.bRcv01	:= stControl.nRcvBoolData.1;
		stHstData.bRcv02	:= stControl.nRcvBoolData.2;
		stHstData.bRcv03	:= stControl.nRcvBoolData.3;
		stHstData.bRcv04	:= stControl.nRcvBoolData.4;
		stHstData.bRcv05	:= stControl.nRcvBoolData.5;
		stHstData.bRcv06	:= stControl.nRcvBoolData.6;
		stHstData.bRcv07	:= stControl.nRcvBoolData.7;
		stHstData.bRcv08	:= stControl.nRcvBoolData.8;  
		stHstData.bRcv09	:= stControl.nRcvBoolData.9;  
		stHstData.bRcv10	:= stControl.nRcvBoolData.10;  
		stHstData.bRcv11	:= stControl.nRcvBoolData.11;  
		stHstData.bRcv12	:= stControl.nRcvBoolData.12; 
		stHstData.bRcv13	:= stControl.nRcvBoolData.13; 
		stHstData.bRcv14	:= stControl.nRcvBoolData.14; 
		stHstData.bRcv15	:= stControl.nRcvBoolData.15;	
		stHstData.nRcv00	:= stControl.nRcvInt00;
		stHstData.nRcv01	:= stControl.nRcvInt01;
	END_IF

(* Send data *)
	stStatus.nSendData				:= BOOL_TO_WORD(stHstData.bSubsOn);
	stStatus.nSendSequenceNumber	:= stControl.nRcvSequenceNumber;
	stStatus.nSendCrc 				:= F_CalcCrc16(ADR(stStatus.nSendData), 2, stConfig.nDpDpId, N_POLYNOM);
END_METHOD

METHOD INTERNAL GetControlData
VAR_INPUT
END_VAR
IF pControl <= 0 OR stConfig.bForceMode THEN RETURN; END_IF

// nRcvBoolData
F_Memcpy(ADR(stControl), pControl, 2, stConfig.bSwapProcessData);
// nRcvInt00
F_Memcpy(ADR(stControl) + 2, pControl + 2, 2, stConfig.bSwapProcessData);		
// nRcvInt01
F_Memcpy(ADR(stControl) + 4, pControl + 4, 2, stConfig.bSwapProcessData);			
// nRcvData
F_Memcpy(ADR(stControl) + 6, pControl + 6, 2, stConfig.bSwapProcessData);			
// nRcvSequenceNumber
F_Memcpy(ADR(stControl) + 8, pControl + 8, 2, stConfig.bSwapProcessData);	
// nRcvCrc
F_Memcpy(ADR(stControl) + 10, pControl + 10, 2, stConfig.bSwapProcessData);
END_METHOD

METHOD INTERNAL InitRun : BOOL
VAR_INST
	bInitRun : BOOL := TRUE;
END_VAR
IF NOT bInitRun THEN RETURN; END_IF
bInitRun := FALSE;

IF pControl = 0 OR pStatus = 0 THEN
	ADSLOGSTR(ADSLOG_MSGTYPE_WARN, CONCAT(_sPath, ': %s'), 'Plc address not set.');
END_IF

_TonTimeout.PT := REAL_TO_TIME(stConfig.fTimeout);
END_METHOD

METHOD INTERNAL SetStatusData
VAR_INPUT
END_VAR
IF pStatus <= 0 THEN RETURN; END_IF


// nSendData
F_Memcpy(pStatus, ADR(stStatus), 2, stConfig.bSwapProcessData);				
// nSendSequenceNumber
F_Memcpy(pStatus + 2, ADR(stStatus) + 2, 2, stConfig.bSwapProcessData);
// nSendCrc
F_Memcpy(pStatus + 4, ADR(stStatus) + 4, 2, stConfig.bSwapProcessData);
END_METHOD

METHOD PRIVATE SimLogic
VAR_INPUT
END_VAR
(* No error or substitude values in sim mode *)
	stHstData.bError 	:= FALSE;
	stHstData.bSubsOn	:= FALSE;

(* Get safety values *)
	stHstData.bRcv00	:= stControl.nRcvBoolData.0;
	stHstData.bRcv01	:= stControl.nRcvBoolData.1;
	stHstData.bRcv02	:= stControl.nRcvBoolData.2;
	stHstData.bRcv03	:= stControl.nRcvBoolData.3;
	stHstData.bRcv04	:= stControl.nRcvBoolData.4;
	stHstData.bRcv05	:= stControl.nRcvBoolData.5;
	stHstData.bRcv06	:= stControl.nRcvBoolData.6;
	stHstData.bRcv07	:= stControl.nRcvBoolData.7;
	stHstData.bRcv08	:= stControl.nRcvBoolData.8;  
	stHstData.bRcv09	:= stControl.nRcvBoolData.9;  
	stHstData.bRcv10	:= stControl.nRcvBoolData.10;  
	stHstData.bRcv11	:= stControl.nRcvBoolData.11;  
	stHstData.bRcv12	:= stControl.nRcvBoolData.12; 
	stHstData.bRcv13	:= stControl.nRcvBoolData.13; 
	stHstData.bRcv14	:= stControl.nRcvBoolData.14; 
	stHstData.bRcv15	:= stControl.nRcvBoolData.15;	
	stHstData.nRcv00	:= stControl.nRcvInt00;
	stHstData.nRcv01	:= stControl.nRcvInt01;

(* Send data *)
	stStatus.nSendData				:= 16#80;
	stStatus.nSendSequenceNumber	:= stControl.nRcvSequenceNumber;
	stStatus.nSendCrc 				:= F_CalcCrc16(ADR(stStatus.nSendData), 2, stConfig.nDpDpId, N_POLYNOM);
END_METHOD

END_FUNCTION_BLOCK

// Devices/Siemens_SendDp/FB_Siemens_SendDp
(*
FB_Siemens_SendDp simulates the funcitionalty of a Siemens PN/PN coupler SENDDP safety-related communication.

Disclaimer: This simulation is an independent project and is not affiliated with, endorsed by, or approved by Siemens. All rights to the Siemens brand name and trademarks remain the property of the manufacturer.
Furthermore, no guarantee is given for the completeness of the functional scope or the error-free operation of the simulation. Users should be aware that deviations from the actual product may occur.
*)

{attribute 'reflection'} 
FUNCTION_BLOCK FB_Siemens_SendDp EXTENDS FB_Base
VAR_INPUT
	pControl 			: PVOID; //Pocess data from fieldbus. Size must be >= stControl.
	pStatus 			: PVOID; //Pocess data to fieldbus. Size must be >= stStatus.
	stControl				: ST_Siemens_SendDp_Control; 	
	stConfig 			: ST_Siemens_SendDp_Config;
	
	stDevData			: ST_Siemens_SendDp_DevData;
END_VAR

VAR_OUTPUT
	stStatus			: ST_Siemens_SendDp_Status; 	

	stHstData			: ST_Siemens_SendDp_HstData;
END_VAR

VAR
    {attribute 'instance-path'} 
    {attribute 'noinit'} 
    _sPath 				: STRING; 
	
	_nLastSequenceNumber	: WORD;
	_nSendSequenceNumber	: WORD;
	_nCalculatedCrc		: WORD;	
	_TonTimeout			: TON;
END_VAR

VAR CONSTANT
	POLYNOM			: WORD := 16#4EAB;
END_VAR

SUPER^();
InitRun();
GetControlData();
Cycle();
SetStatusData();

METHOD PRIVATE Cycle
(* Simplified communication when using PLCSIM Adv. *)
	IF OC_Core.GVL_Core.fbSystem.eControllerType = E_ControllerType.PlcSimAdvanced THEN
		SimLogic();
		RETURN;
	END_IF

(* Calculate received crc *)
	_nCalculatedCrc := F_CalcCrc16(ADR(stControl), 2, stConfig.nDpDpId, POLYNOM);

(* Restart timer, if sequence number has changed *)
	IF stControl.nRcvSequenceNumber <> _nLastSequenceNumber THEN
		_TonTimeout.IN		:= FALSE;
		_nLastSequenceNumber := stControl.nRcvSequenceNumber;
		stHstData.bError	:= FALSE;
		stHstData.bSubsOn	:= FALSE;
	ELSE
		_TonTimeout.IN		:= TRUE;
	END_IF

(* Check if timer has expired *)
	_TonTimeout();
	
	IF _TonTimeout.Q	THEN
		_TonTimeout.IN		:= FALSE;
		_nSendSequenceNumber := 0;
		stHstData.bError	:= TRUE;
		stHstData.bSubsOn	:= TRUE;
	END_IF

(* compare received crc value with calculated crc *)
	IF stControl.nRcvCrc = _nCalculatedCrc THEN
		IF _nSendSequenceNumber = stControl.nRcvSequenceNumber THEN
			IF _nSendSequenceNumber = 0 THEN
				_nSendSequenceNumber := 1;
			ELSE
				_nSendSequenceNumber := _nSendSequenceNumber + 1;
			END_IF
		END_IF
	END_IF

(* Limit sequence number to 32767 *)
	IF _nSendSequenceNumber > 32767 THEN
		_nSendSequenceNumber := 1;
	END_IF

(* Send data *)
	stStatus.nSendBoolData.0 		:= stDevData.bSend00;
	stStatus.nSendBoolData.1 		:= stDevData.bSend01;
	stStatus.nSendBoolData.2 		:= stDevData.bSend02;
	stStatus.nSendBoolData.3 		:= stDevData.bSend03;
	stStatus.nSendBoolData.4 		:= stDevData.bSend04;
	stStatus.nSendBoolData.5 		:= stDevData.bSend05;
	stStatus.nSendBoolData.6 		:= stDevData.bSend06;
	stStatus.nSendBoolData.7 		:= stDevData.bSend07;
	stStatus.nSendBoolData.8 		:= stDevData.bSend08;
	stStatus.nSendBoolData.9 		:= stDevData.bSend09;
	stStatus.nSendBoolData.10 		:= stDevData.bSend10;
	stStatus.nSendBoolData.11 		:= stDevData.bSend11;
	stStatus.nSendBoolData.12 		:= stDevData.bSend12;
	stStatus.nSendBoolData.13 		:= stDevData.bSend13;
	stStatus.nSendBoolData.14 		:= stDevData.bSend14;
	stStatus.nSendBoolData.15 		:= stDevData.bSend15;
	stStatus.nSendInt00				:= stDevData.nSend00;
	stStatus.nSendInt01				:= stDevData.nSend01;
	stStatus.nSendData				:= BOOL_TO_WORD(stHstData.bSubsOn);
	stStatus.nSendSequenceNumber 	:= _nSendSequenceNumber;
	stStatus.nSendCrc 				:= F_CalcCrc16(ADR(stStatus), 8, stConfig.nDpDpId, POLYNOM);
END_METHOD

METHOD INTERNAL GetControlData
VAR_INPUT
END_VAR
IF pControl <= 0 OR stConfig.bForceMode THEN RETURN; END_IF

// nRcvData
F_Memcpy(ADR(stControl), pControl, 2, stConfig.bSwapProcessData);
// nRcvSequenceNumber
F_Memcpy(ADR(stControl) + 2, pControl + 2, 2, stConfig.bSwapProcessData);
// nRcvCrc
F_Memcpy(ADR(stControl) + 4, pControl + 4, 2, stConfig.bSwapProcessData);
END_METHOD

METHOD INTERNAL InitRun : BOOL
VAR_INST
	bInitRun : BOOL := TRUE;
END_VAR
IF NOT bInitRun THEN RETURN; END_IF
bInitRun := FALSE;

IF pControl = 0 OR pStatus = 0 THEN
	ADSLOGSTR(ADSLOG_MSGTYPE_WARN, CONCAT(_sPath, ': %s'), 'Plc address not set.');
END_IF

_TonTimeout.PT := REAL_TO_TIME(stConfig.fTimeout);
END_METHOD

METHOD INTERNAL SetStatusData
VAR_INPUT
END_VAR
IF pStatus <= 0 THEN RETURN; END_IF

// nSendBoolData
F_Memcpy(pStatus, ADR(stStatus), 2, stConfig.bSwapProcessData);
// nSendInt00
F_Memcpy(pStatus + 2, ADR(stStatus) + 2, 2, stConfig.bSwapProcessData);		
// nSendInt01
F_Memcpy(pStatus + 4, ADR(stStatus) + 4, 2, stConfig.bSwapProcessData);		
// nSendData
F_Memcpy(pStatus + 6, ADR(stStatus) + 6, 2, stConfig.bSwapProcessData);	
// nSendSequenceNumber
F_Memcpy(pStatus + 8, ADR(stStatus) + 8, 2, stConfig.bSwapProcessData);
// nSendCrc
F_Memcpy(pStatus + 10, ADR(stStatus) + 10, 2, stConfig.bSwapProcessData);
END_METHOD

METHOD PRIVATE SimLogic
VAR_INPUT
END_VAR
(* No error or substitude values in sim mode *)
	stHstData.bError 	:= FALSE;
	stHstData.bSubsOn	:= FALSE;

(* Send data *)
	stStatus.nSendBoolData.0 		:= stDevData.bSend00;
	stStatus.nSendBoolData.1 		:= stDevData.bSend01;
	stStatus.nSendBoolData.2 		:= stDevData.bSend02;
	stStatus.nSendBoolData.3 		:= stDevData.bSend03;
	stStatus.nSendBoolData.4 		:= stDevData.bSend04;
	stStatus.nSendBoolData.5 		:= stDevData.bSend05;
	stStatus.nSendBoolData.6 		:= stDevData.bSend06;
	stStatus.nSendBoolData.7 		:= stDevData.bSend07;
	stStatus.nSendBoolData.8 		:= stDevData.bSend08;
	stStatus.nSendBoolData.9 		:= stDevData.bSend09;
	stStatus.nSendBoolData.10 		:= stDevData.bSend10;
	stStatus.nSendBoolData.11 		:= stDevData.bSend11;
	stStatus.nSendBoolData.12 		:= stDevData.bSend12;
	stStatus.nSendBoolData.13 		:= stDevData.bSend13;
	stStatus.nSendBoolData.14 		:= stDevData.bSend14;
	stStatus.nSendBoolData.15 		:= stDevData.bSend15;
	stStatus.nSendInt00				:= stDevData.nSend00;
	stStatus.nSendInt01				:= stDevData.nSend01;
	stStatus.nSendData				:= 16#80;
	stStatus.nSendSequenceNumber 	:= 16#FFFF;
	stStatus.nSendCrc 				:= F_CalcCrc16(ADR(stStatus), 8, stConfig.nDpDpId, POLYNOM);
END_METHOD

END_FUNCTION_BLOCK
